LIN {X 0,Y 397.089,Z 381.624,A -85,B 0,C 180,E1 -11120.42,E2 -11120.42} C_VEL
LIN {X 0,Y 397.097,Z 381.645,A -85,B 0,C 180,E1 -11123.005,E2 -11123.005} C_VEL
LIN {X 0,Y 397.114,Z 381.63,A -85,B 0,C 180,E1 -11126.727,E2 -11126.727} C_VEL
LIN {X 0,Y 397.12,Z 381.643,A -85,B 0,C 180,E1 -11130.295,E2 -11130.295} C_VEL
LIN {X 0,Y 397.076,Z 381.648,A -85,B 0,C 180,E1 -11133.737,E2 -11133.737} C_VEL
LIN {X 0,Y 397.149,Z 381.85,A -85,B 0,C 180,E1 -11134.804,E2 -11134.804} C_VEL
LIN {X 0,Y 398.52,Z 387.762,A -85,B 0,C 180,E1 -11136.032,E2 -11136.032} C_VEL
LIN {X 0,Y 406.526,Z 408.883,A -85,B 0,C 180,E1 -11136.981,E2 -11136.981} C_VEL
LIN {X 0,Y 404.185,Z 503.873,A -85,B 0,C 180,E1 -11139.084,E2 -11139.084} C_VEL
LIN {X 0,Y 403.629,Z 530.739,A -85,B 0,C 180,E1 -11139.707,E2 -11139.707} C_VEL
LIN {X 0,Y 403.24,Z 546.56,A -85,B 0,C 180,E1 -11140.291,E2 -11140.291} C_VEL
LIN {X 0,Y 402.743,Z 560.989,A -85,B 0,C 180,E1 -11141.034,E2 -11141.034} C_VEL
LIN {X 0,Y 402.067,Z 574.399,A -85,B 0,C 180,E1 -11141.925,E2 -11141.925} C_VEL
LIN {X 0,Y 401.478,Z 586.705,A -85,B 0,C 180,E1 -11142.949,E2 -11142.949} C_VEL
LIN {X 0,Y 400.667,Z 599.243,A -85,B 0,C 180,E1 -11144.224,E2 -11144.224} C_VEL
LIN {X 0,Y 399.964,Z 610.425,A -85,B 0,C 180,E1 -11145.604,E2 -11145.604} C_VEL
LIN {X 0,Y 399.225,Z 620.083,A -85,B 0,C 180,E1 -11147.029,E2 -11147.029} C_VEL
LIN {X 0,Y 398.678,Z 628.735,A -85,B 0,C 180,E1 -11148.561,E2 -11148.561} C_VEL
LIN {X 0,Y 398.179,Z 637.057,A -85,B 0,C 180,E1 -11150.347,E2 -11150.347} C_VEL
LIN {X 0,Y 397.823,Z 642.855,A -85,B 0,C 180,E1 -11151.875,E2 -11151.875} C_VEL
LIN {X 0,Y 397.588,Z 647.629,A -85,B 0,C 180,E1 -11153.402,E2 -11153.402} C_VEL
LIN {X 0,Y 397.252,Z 651.509,A -85,B 0,C 180,E1 -11154.925,E2 -11154.925} C_VEL
LIN {X 0,Y 397.11,Z 653.565,A -85,B 0,C 180,E1 -11155.94,E2 -11155.94} C_VEL
LIN {X 0,Y 397.246,Z 655.212,A -85,B 0,C 180,E1 -11156.957,E2 -11156.957} C_VEL
LIN {X 0,Y 397.195,Z 657.492,A -85,B 0,C 180,E1 -11158.986,E2 -11158.986} C_VEL
LIN {X 0,Y 397.255,Z 658.37,A -85,B 0,C 180,E1 -11161.014,E2 -11161.014} C_VEL
LIN {X 0,Y 397.563,Z 657.822,A -85,B 0,C 180,E1 -11163.04,E2 -11163.04} C_VEL
LIN {X 0,Y 397.875,Z 655.889,A -85,B 0,C 180,E1 -11165.067,E2 -11165.067} C_VEL
LIN {X 0,Y 398.072,Z 654.383,A -85,B 0,C 180,E1 -11166.081,E2 -11166.081} C_VEL
LIN {X 0,Y 398.686,Z 651.307,A -85,B 0,C 180,E1 -11167.597,E2 -11167.597} C_VEL
LIN {X 0,Y 399.26,Z 646.78,A -85,B 0,C 180,E1 -11169.32,E2 -11169.32} C_VEL
LIN {X 0,Y 400.073,Z 640.589,A -85,B 0,C 180,E1 -11171.142,E2 -11171.142} C_VEL
LIN {X 0,Y 401.076,Z 633.002,A -85,B 0,C 180,E1 -11172.91,E2 -11172.91} C_VEL
LIN {X 0,Y 402.077,Z 624.982,A -85,B 0,C 180,E1 -11174.423,E2 -11174.423} C_VEL
LIN {X 0,Y 403.151,Z 615.267,A -85,B 0,C 180,E1 -11175.936,E2 -11175.936} C_VEL
LIN {X 0,Y 404.407,Z 603.369,A -85,B 0,C 180,E1 -11177.444,E2 -11177.444} C_VEL
LIN {X 0,Y 405.456,Z 591.237,A -85,B 0,C 180,E1 -11178.703,E2 -11178.703} C_VEL
LIN {X 0,Y 406.37,Z 579.301,A -85,B 0,C 180,E1 -11179.709,E2 -11179.709} C_VEL
LIN {X 0,Y 407.245,Z 566.122,A -85,B 0,C 180,E1 -11180.602,E2 -11180.602} C_VEL
LIN {X 0,Y 407.975,Z 552.389,A -85,B 0,C 180,E1 -11181.325,E2 -11181.325} C_VEL
LIN {X 0,Y 408.412,Z 537.34,A -85,B 0,C 180,E1 -11181.913,E2 -11181.913} C_VEL
LIN {X 0,Y 410.593,Z 491.111,A -85,B 0,C 180,E1 -11183.217,E2 -11183.217} C_VEL
LIN {X 0,Y 415.197,Z 422.298,A -85,B 0,C 180,E1 -11185.198,E2 -11185.198} C_VEL
LIN {X 0,Y 414.865,Z 420.892,A -85,B 0,C 180,E1 -11185.293,E2 -11185.293} C_VEL
LIN {X 0,Y 408.921,Z 410.512,A -85,B 0,C 180,E1 -11186.453,E2 -11186.453} C_VEL
LIN {X 0,Y 405.011,Z 404.284,A -85,B 0,C 180,E1 -11187.301,E2 -11187.301} C_VEL
LIN {X 0,Y 403.247,Z 398.209,A -85,B 0,C 180,E1 -11189.782,E2 -11189.782} C_VEL
LIN {X 0,Y 401.316,Z 392.497,A -85,B 0,C 180,E1 -11192.795,E2 -11192.795} C_VEL
LIN {X 0,Y 400.112,Z 388.952,A -85,B 0,C 180,E1 -11195.426,E2 -11195.426} C_VEL
LIN {X 0,Y 399.12,Z 386.996,A -85,B 0,C 180,E1 -11198.047,E2 -11198.047} C_VEL
LIN {X 0,Y 398.976,Z 386.521,A -85,B 0,C 180,E1 -11199.356,E2 -11199.356} C_VEL
LIN {X 0,Y 398.969,Z 386.501,A -85,B 0,C 180,E1 -11200.758,E2 -11200.758} C_VEL
LIN {X 0,Y 399.211,Z 387.025,A -85,B 0,C 180,E1 -11202.318,E2 -11202.318} C_VEL
LIN {X 0,Y 400.18,Z 388.851,A -85,B 0,C 180,E1 -11204.626,E2 -11204.626} C_VEL
LIN {X 0,Y 401.605,Z 392.32,A -85,B 0,C 180,E1 -11206.96,E2 -11206.96} C_VEL
LIN {X 0,Y 403.759,Z 397.673,A -85,B 0,C 180,E1 -11209.425,E2 -11209.425} C_VEL
LIN {X 0,Y 405.909,Z 403.521,A -85,B 0,C 180,E1 -11211.44,E2 -11211.44} C_VEL
LIN {X 0,Y 408.329,Z 411.193,A -85,B 0,C 180,E1 -11213.575,E2 -11213.575} C_VEL
LIN {X 0,Y 410.262,Z 418.651,A -85,B 0,C 180,E1 -11215.312,E2 -11215.312} C_VEL
LIN {X 0,Y 411.173,Z 423.227,A -85,B 0,C 180,E1 -11216.253,E2 -11216.253} C_VEL
LIN {X 0,Y 410.818,Z 426.707,A -85,B 0,C 180,E1 -11216.808,E2 -11216.808} C_VEL
LIN {X 0,Y 407.511,Z 447.425,A -85,B 0,C 180,E1 -11219.787,E2 -11219.787} C_VEL
LIN {X 0,Y 407.066,Z 451.037,A -85,B 0,C 180,E1 -11220.274,E2 -11220.274} C_VEL
LIN {X 0,Y 409.714,Z 468.904,A -85,B 0,C 180,E1 -11221.206,E2 -11221.206} C_VEL
LIN {X 0,Y 411.359,Z 484.62,A -85,B 0,C 180,E1 -11221.892,E2 -11221.892} C_VEL
LIN {X 0,Y 412.406,Z 501.199,A -85,B 0,C 180,E1 -11222.511,E2 -11222.511} C_VEL
LIN {X 0,Y 410.024,Z 555.027,A -85,B 0,C 180,E1 -11223.842,E2 -11223.842} C_VEL
LIN {X 0,Y 408.208,Z 641.314,A -85,B 0,C 180,E1 -11225.389,E2 -11225.389} C_VEL
LIN {X 0,Y 407.512,Z 656.884,A -85,B 0,C 180,E1 -11225.87,E2 -11225.87} C_VEL
LIN {X 0,Y 406.506,Z 672.375,A -85,B 0,C 180,E1 -11226.568,E2 -11226.568} C_VEL
LIN {X 0,Y 405.354,Z 686.866,A -85,B 0,C 180,E1 -11227.442,E2 -11227.442} C_VEL
LIN {X 0,Y 404.081,Z 700.048,A -85,B 0,C 180,E1 -11228.442,E2 -11228.442} C_VEL
LIN {X 0,Y 402.632,Z 713.43,A -85,B 0,C 180,E1 -11229.7,E2 -11229.7} C_VEL
LIN {X 0,Y 401.283,Z 725.191,A -85,B 0,C 180,E1 -11231.04,E2 -11231.04} C_VEL
LIN {X 0,Y 399.941,Z 736.663,A -85,B 0,C 180,E1 -11232.617,E2 -11232.617} C_VEL
LIN {X 0,Y 398.771,Z 747.384,A -85,B 0,C 180,E1 -11234.408,E2 -11234.408} C_VEL
LIN {X 0,Y 397.723,Z 756.499,A -85,B 0,C 180,E1 -11236.246,E2 -11236.246} C_VEL
LIN {X 0,Y 397.007,Z 764.608,A -85,B 0,C 180,E1 -11238.252,E2 -11238.252} C_VEL
LIN {X 0,Y 396.384,Z 771.265,A -85,B 0,C 180,E1 -11240.302,E2 -11240.302} C_VEL
LIN {X 0,Y 396.048,Z 776.466,A -85,B 0,C 180,E1 -11242.35,E2 -11242.35} C_VEL
LIN {X 0,Y 395.949,Z 779.458,A -85,B 0,C 180,E1 -11243.885,E2 -11243.885} C_VEL
LIN {X 0,Y 395.81,Z 782.389,A -85,B 0,C 180,E1 -11245.926,E2 -11245.926} C_VEL
LIN {X 0,Y 395.823,Z 784.133,A -85,B 0,C 180,E1 -11247.963,E2 -11247.963} C_VEL
LIN {X 0,Y 395.812,Z 784.728,A -85,B 0,C 180,E1 -11249.998,E2 -11249.998} C_VEL
LIN {X 0,Y 395.839,Z 784.13,A -85,B 0,C 180,E1 -11252.033,E2 -11252.033} C_VEL
LIN {X 0,Y 395.814,Z 782.381,A -85,B 0,C 180,E1 -11254.071,E2 -11254.071} C_VEL
LIN {X 0,Y 395.911,Z 779.235,A -85,B 0,C 180,E1 -11256.238,E2 -11256.238} C_VEL
LIN {X 0,Y 396.129,Z 775.273,A -85,B 0,C 180,E1 -11258.158,E2 -11258.158} C_VEL
LIN {X 0,Y 396.472,Z 769.727,A -85,B 0,C 180,E1 -11260.209,E2 -11260.209} C_VEL
LIN {X 0,Y 397.186,Z 762.664,A -85,B 0,C 180,E1 -11262.257,E2 -11262.257} C_VEL
LIN {X 0,Y 397.854,Z 755.214,A -85,B 0,C 180,E1 -11264.029,E2 -11264.029} C_VEL
LIN {X 0,Y 398.858,Z 745.957,A -85,B 0,C 180,E1 -11265.848,E2 -11265.848} C_VEL
LIN {X 0,Y 399.907,Z 736.641,A -85,B 0,C 180,E1 -11267.381,E2 -11267.381} C_VEL
LIN {X 0,Y 401.058,Z 727.016,A -85,B 0,C 180,E1 -11268.716,E2 -11268.716} C_VEL
LIN {X 0,Y 402.339,Z 715.741,A -85,B 0,C 180,E1 -11270.046,E2 -11270.046} C_VEL
LIN {X 0,Y 403.723,Z 702.844,A -85,B 0,C 180,E1 -11271.307,E2 -11271.307} C_VEL
LIN {X 0,Y 404.986,Z 690.311,A -85,B 0,C 180,E1 -11272.308,E2 -11272.308} C_VEL
LIN {X 0,Y 406.228,Z 675.667,A -85,B 0,C 180,E1 -11273.243,E2 -11273.243} C_VEL
LIN {X 0,Y 407.212,Z 661.406,A -85,B 0,C 180,E1 -11273.94,E2 -11273.94} C_VEL
LIN {X 0,Y 407.963,Z 646.864,A -85,B 0,C 180,E1 -11274.454,E2 -11274.454} C_VEL
LIN {X 0,Y 408.469,Z 630.141,A -85,B 0,C 180,E1 -11274.828,E2 -11274.828} C_VEL
LIN {X 0,Y 410.947,Z 500.531,A -85,B 0,C 180,E1 -11277.127,E2 -11277.127} C_VEL
LIN {X 0,Y 407.131,Z 470.69,A -85,B 0,C 180,E1 -11277.985,E2 -11277.985} C_VEL
LIN {X 0,Y 406.3,Z 464.366,A -85,B 0,C 180,E1 -11278.213,E2 -11278.213} C_VEL
LIN {X 0,Y 405.055,Z 449.15,A -85,B 0,C 180,E1 -11279.028,E2 -11279.028} C_VEL
LIN {X 0,Y 407.471,Z 422.518,A -85,B 0,C 180,E1 -11282.32,E2 -11282.32} C_VEL
LIN {X 0,Y 407.781,Z 419.227,A -85,B 0,C 180,E1 -11282.732,E2 -11282.732} C_VEL
LIN {X 0,Y 404.459,Z 406.774,A -85,B 0,C 180,E1 -11284.594,E2 -11284.594} C_VEL
LIN {X 0,Y 398.163,Z 385.398,A -85,B 0,C 180,E1 -11287.984,E2 -11287.984} C_VEL
LIN {X 0,Y 397.122,Z 381.788,A -85,B 0,C 180,E1 -11288.623,E2 -11288.623} C_VEL
LIN {X 0,Y 397.045,Z 381.654,A -85,B 0,C 180,E1 -11292.267,E2 -11292.267} C_VEL
LIN {X 0,Y 397.072,Z 381.648,A -85,B 0,C 180,E1 -11295.068,E2 -11295.068} C_VEL
LIN {X 0,Y 397.038,Z 381.618,A -85,B 0,C 180,E1 -11298.023,E2 -11298.023} C_VEL
LIN {X 0,Y 397.076,Z 381.648,A -85,B 0,C 180,E1 -11301.722,E2 -11301.722} C_VEL
LIN {X 0,Y 397.102,Z 381.606,A -85,B 0,C 180,E1 -11305.505,E2 -11305.505} C_VEL
LIN {X 0,Y 397.063,Z 381.648,A -85,B 0,C 180,E1 -11309.116,E2 -11309.116} C_VEL
LIN {X 0,Y 397.064,Z 381.647,A -85,B 0,C 180,E1 -11312.246,E2 -11312.246} C_VEL
LIN {X 0,Y 397.089,Z 381.633,A -85,B 0,C 180,E1 -11314.864,E2 -11314.864} C_VEL
LIN {X 0,Y 397.08,Z 381.65,A -85,B 0,C 180,E1 -11318.181,E2 -11318.181} C_VEL
LIN {X 0,Y 397.098,Z 381.641,A -85,B 0,C 180,E1 -11321.424,E2 -11321.424} C_VEL
LIN {X 0,Y 397.108,Z 381.631,A -85,B 0,C 180,E1 -11324.605,E2 -11324.605} C_VEL
LIN {X 0,Y 397.202,Z 381.631,A -85,B 0,C 180,E1 -11327.741,E2 -11327.741} C_VEL
LIN {X 0,Y 397.212,Z 381.618,A -85,B 0,C 180,E1 -11330.837,E2 -11330.837} C_VEL
LIN {X 0,Y 397.299,Z 381.618,A -85,B 0,C 180,E1 -11333.907,E2 -11333.907} C_VEL
LIN {X 0,Y 397.427,Z 381.601,A -85,B 0,C 180,E1 -11337.973,E2 -11337.973} C_VEL
LIN {X 0,Y 397.424,Z 381.591,A -85,B 0,C 180,E1 -11342.027,E2 -11342.027} C_VEL
LIN {X 0,Y 397.305,Z 381.606,A -85,B 0,C 180,E1 -11346.708,E2 -11346.708} C_VEL
LIN {X 0,Y 397.217,Z 381.629,A -85,B 0,C 180,E1 -11349.163,E2 -11349.163} C_VEL
LIN {X 0,Y 397.202,Z 381.616,A -85,B 0,C 180,E1 -11352.259,E2 -11352.259} C_VEL
LIN {X 0,Y 397.162,Z 381.629,A -85,B 0,C 180,E1 -11355.393,E2 -11355.393} C_VEL
LIN {X 0,Y 397.143,Z 381.638,A -85,B 0,C 180,E1 -11358.574,E2 -11358.574} C_VEL
LIN {X 0,Y 397.08,Z 381.638,A -85,B 0,C 180,E1 -11361.82,E2 -11361.82} C_VEL
LIN {X 0,Y 397.087,Z 381.636,A -85,B 0,C 180,E1 -11365.136,E2 -11365.136} C_VEL
LIN {X 0,Y 397.048,Z 381.648,A -85,B 0,C 180,E1 -11368.55,E2 -11368.55} C_VEL
LIN {X 0,Y 397.064,Z 381.649,A -85,B 0,C 180,E1 -11371.836,E2 -11371.836} C_VEL
LIN {X 0,Y 397.104,Z 381.649,A -85,B 0,C 180,E1 -11374.496,E2 -11374.496} C_VEL
LIN {X 0,Y 397.077,Z 381.623,A -85,B 0,C 180,E1 -11378.278,E2 -11378.278} C_VEL
LIN {X 0,Y 397.035,Z 381.648,A -85,B 0,C 180,E1 -11380.916,E2 -11380.916} C_VEL
LIN {X 0,Y 397.075,Z 381.635,A -85,B 0,C 180,E1 -11383.652,E2 -11383.652} C_VEL
LIN {X 0,Y 397.08,Z 381.631,A -85,B 0,C 180,E1 -11386.525,E2 -11386.525} C_VEL
LIN {X 0,Y 397.13,Z 381.847,A -85,B 0,C 180,E1 -11389.321,E2 -11389.321} C_VEL
LIN {X 0,Y 399.981,Z 390.021,A -85,B 0,C 180,E1 -11390.764,E2 -11390.764} C_VEL
LIN {X 0,Y 405.051,Z 405.352,A -85,B 0,C 180,E1 -11393.294,E2 -11393.294} C_VEL
LIN {X 0,Y 409.446,Z 421.082,A -85,B 0,C 180,E1 -11395.744,E2 -11395.744} C_VEL
LIN {X 0,Y 409.79,Z 422.39,A -85,B 0,C 180,E1 -11395.94,E2 -11395.94} C_VEL
LIN {X 0,Y 409.04,Z 433.785,A -85,B 0,C 180,E1 -11397.342,E2 -11397.342} C_VEL
LIN {X 0,Y 407.476,Z 457.22,A -85,B 0,C 180,E1 -11400.133,E2 -11400.133} C_VEL
LIN {X 0,Y 406.73,Z 471.528,A -85,B 0,C 180,E1 -11401.751,E2 -11401.751} C_VEL
LIN {X 0,Y 411.653,Z 502.312,A -85,B 0,C 180,E1 -11402.733,E2 -11402.733} C_VEL
LIN {X 0,Y 408.849,Z 639.721,A -85,B 0,C 180,E1 -11405.197,E2 -11405.197} C_VEL
LIN {X 0,Y 408.137,Z 655.686,A -85,B 0,C 180,E1 -11405.665,E2 -11405.665} C_VEL
LIN {X 0,Y 407.159,Z 670.76,A -85,B 0,C 180,E1 -11406.317,E2 -11406.317} C_VEL
LIN {X 0,Y 406.104,Z 684.154,A -85,B 0,C 180,E1 -11407.086,E2 -11407.086} C_VEL
LIN {X 0,Y 404.743,Z 697.956,A -85,B 0,C 180,E1 -11408.081,E2 -11408.081} C_VEL
LIN {X 0,Y 403.391,Z 710.624,A -85,B 0,C 180,E1 -11409.21,E2 -11409.21} C_VEL
LIN {X 0,Y 402.084,Z 722.357,A -85,B 0,C 180,E1 -11410.473,E2 -11410.473} C_VEL
LIN {X 0,Y 400.806,Z 733.238,A -85,B 0,C 180,E1 -11411.868,E2 -11411.868} C_VEL
LIN {X 0,Y 399.525,Z 743.27,A -85,B 0,C 180,E1 -11413.392,E2 -11413.392} C_VEL
LIN {X 0,Y 398.336,Z 753.073,A -85,B 0,C 180,E1 -11415.179,E2 -11415.179} C_VEL
LIN {X 0,Y 397.433,Z 761.858,A -85,B 0,C 180,E1 -11417.133,E2 -11417.133} C_VEL
LIN {X 0,Y 396.459,Z 764.8,A -85,B 0,C 180,E1 -11417.861,E2 -11417.861} C_VEL
LIN {X 0,Y 393.176,Z 769.275,A -85,B 0,C 180,E1 -11419.057,E2 -11419.057} C_VEL
LIN {X 0,Y 389.974,Z 773.232,A -85,B 0,C 180,E1 -11420.305,E2 -11420.305} C_VEL
LIN {X 0,Y 389.137,Z 775.372,A -85,B 0,C 180,E1 -11421.103,E2 -11421.103} C_VEL
LIN {X 0,Y 388.85,Z 779.022,A -85,B 0,C 180,E1 -11422.733,E2 -11422.733} C_VEL
LIN {X 0,Y 388.697,Z 782.564,A -85,B 0,C 180,E1 -11424.815,E2 -11424.815} C_VEL
LIN {X 0,Y 388.59,Z 784.906,A -85,B 0,C 180,E1 -11426.891,E2 -11426.891} C_VEL
LIN {X 0,Y 388.652,Z 786.099,A -85,B 0,C 180,E1 -11428.965,E2 -11428.965} C_VEL
LIN {X 0,Y 388.653,Z 786.114,A -85,B 0,C 180,E1 -11431.038,E2 -11431.038} C_VEL
LIN {X 0,Y 388.591,Z 784.981,A -85,B 0,C 180,E1 -11433.112,E2 -11433.112} C_VEL
LIN {X 0,Y 388.709,Z 782.697,A -85,B 0,C 180,E1 -11435.188,E2 -11435.188} C_VEL
LIN {X 0,Y 388.919,Z 779.209,A -85,B 0,C 180,E1 -11437.269,E2 -11437.269} C_VEL
LIN {X 0,Y 389.212,Z 774.436,A -85,B 0,C 180,E1 -11439.354,E2 -11439.354} C_VEL
LIN {X 0,Y 389.809,Z 768.258,A -85,B 0,C 180,E1 -11441.44,E2 -11441.44} C_VEL
LIN {X 0,Y 390.607,Z 760.487,A -85,B 0,C 180,E1 -11443.528,E2 -11443.528} C_VEL
LIN {X 0,Y 391.54,Z 752.198,A -85,B 0,C 180,E1 -11445.354,E2 -11445.354} C_VEL
LIN {X 0,Y 392.795,Z 742.215,A -85,B 0,C 180,E1 -11447.172,E2 -11447.172} C_VEL
LIN {X 0,Y 394.141,Z 732.023,A -85,B 0,C 180,E1 -11448.722,E2 -11448.722} C_VEL
LIN {X 0,Y 395.612,Z 719.815,A -85,B 0,C 180,E1 -11450.27,E2 -11450.27} C_VEL
LIN {X 0,Y 397.133,Z 707.618,A -85,B 0,C 180,E1 -11451.545,E2 -11451.545} C_VEL
LIN {X 0,Y 398.532,Z 694.315,A -85,B 0,C 180,E1 -11452.692,E2 -11452.692} C_VEL
LIN {X 0,Y 399.989,Z 679.521,A -85,B 0,C 180,E1 -11453.7,E2 -11453.7} C_VEL
LIN {X 0,Y 401.097,Z 664.893,A -85,B 0,C 180,E1 -11454.472,E2 -11454.472} C_VEL
LIN {X 0,Y 402.017,Z 649.798,A -85,B 0,C 180,E1 -11455.05,E2 -11455.05} C_VEL
LIN {X 0,Y 402.559,Z 634.992,A -85,B 0,C 180,E1 -11455.429,E2 -11455.429} C_VEL
LIN {X 0,Y 405.369,Z 503.814,A -85,B 0,C 180,E1 -11457.794,E2 -11457.794} C_VEL
LIN {X 0,Y 400.361,Z 472.201,A -85,B 0,C 180,E1 -11458.805,E2 -11458.805} C_VEL
LIN {X 0,Y 400.3,Z 469.804,A -85,B 0,C 180,E1 -11459.02,E2 -11459.02} C_VEL
LIN {X 0,Y 401.927,Z 444.921,A -85,B 0,C 180,E1 -11461.935,E2 -11461.935} C_VEL
LIN {X 0,Y 403.408,Z 425.683,A -85,B 0,C 180,E1 -11464.296,E2 -11464.296} C_VEL
LIN {X 0,Y 400.308,Z 413.802,A -85,B 0,C 180,E1 -11466.138,E2 -11466.138} C_VEL
LIN {X 0,Y 395.695,Z 398.735,A -85,B 0,C 180,E1 -11468.602,E2 -11468.602} C_VEL
LIN {X 0,Y 390.413,Z 384.107,A -85,B 0,C 180,E1 -11471.156,E2 -11471.156} C_VEL
LIN {X 0,Y 390.024,Z 382.673,A -85,B 0,C 180,E1 -11471.479,E2 -11471.479} C_VEL
LIN {X 0,Y 390.008,Z 382.518,A -85,B 0,C 180,E1 -11474.652,E2 -11474.652} C_VEL
LIN {X 0,Y 390.03,Z 382.528,A -85,B 0,C 180,E1 -11477.629,E2 -11477.629} C_VEL
LIN {X 0,Y 390.059,Z 382.504,A -85,B 0,C 180,E1 -11480.904,E2 -11480.904} C_VEL
LIN {X 0,Y 390.072,Z 382.494,A -85,B 0,C 180,E1 -11484.792,E2 -11484.792} C_VEL
LIN {X 0,Y 390.022,Z 382.527,A -85,B 0,C 180,E1 -11488.495,E2 -11488.495} C_VEL
LIN {X 0,Y 390.021,Z 382.528,A -85,B 0,C 180,E1 -11492.003,E2 -11492.003} C_VEL
LIN {X 0,Y 390.076,Z 382.707,A -85,B 0,C 180,E1 -11494.469,E2 -11494.469} C_VEL
LIN {X 0,Y 391.413,Z 388.26,A -85,B 0,C 180,E1 -11495.65,E2 -11495.65} C_VEL
LIN {X 0,Y 399.879,Z 410.632,A -85,B 0,C 180,E1 -11496.682,E2 -11496.682} C_VEL
LIN {X 0,Y 397.151,Z 511.569,A -85,B 0,C 180,E1 -11498.967,E2 -11498.967} C_VEL
LIN {X 0,Y 396.771,Z 533.461,A -85,B 0,C 180,E1 -11499.518,E2 -11499.518} C_VEL
LIN {X 0,Y 396.367,Z 548.749,A -85,B 0,C 180,E1 -11500.114,E2 -11500.114} C_VEL
LIN {X 0,Y 395.802,Z 563.167,A -85,B 0,C 180,E1 -11500.89,E2 -11500.89} C_VEL
LIN {X 0,Y 395.081,Z 577.072,A -85,B 0,C 180,E1 -11501.862,E2 -11501.862} C_VEL
LIN {X 0,Y 394.386,Z 590.414,A -85,B 0,C 180,E1 -11503.034,E2 -11503.034} C_VEL
LIN {X 0,Y 393.54,Z 602.523,A -85,B 0,C 180,E1 -11504.329,E2 -11504.329} C_VEL
LIN {X 0,Y 392.896,Z 613.545,A -85,B 0,C 180,E1 -11505.762,E2 -11505.762} C_VEL
LIN {X 0,Y 392.088,Z 623.491,A -85,B 0,C 180,E1 -11507.316,E2 -11507.316} C_VEL
LIN {X 0,Y 391.581,Z 631.771,A -85,B 0,C 180,E1 -11508.876,E2 -11508.876} C_VEL
LIN {X 0,Y 391.054,Z 639.69,A -85,B 0,C 180,E1 -11510.692,E2 -11510.692} C_VEL
LIN {X 0,Y 390.797,Z 645.268,A -85,B 0,C 180,E1 -11512.248,E2 -11512.248} C_VEL
LIN {X 0,Y 390.406,Z 651.086,A -85,B 0,C 180,E1 -11514.318,E2 -11514.318} C_VEL
LIN {X 0,Y 390.084,Z 654.454,A -85,B 0,C 180,E1 -11515.867,E2 -11515.867} C_VEL
LIN {X 0,Y 390.224,Z 656.151,A -85,B 0,C 180,E1 -11516.903,E2 -11516.903} C_VEL
LIN {X 0,Y 390.172,Z 658.517,A -85,B 0,C 180,E1 -11518.968,E2 -11518.968} C_VEL
LIN {X 0,Y 390.265,Z 659.479,A -85,B 0,C 180,E1 -11521.032,E2 -11521.032} C_VEL
LIN {X 0,Y 390.595,Z 659.016,A -85,B 0,C 180,E1 -11523.094,E2 -11523.094} C_VEL
LIN {X 0,Y 390.933,Z 657.159,A -85,B 0,C 180,E1 -11525.157,E2 -11525.157} C_VEL
LIN {X 0,Y 391.53,Z 653.812,A -85,B 0,C 180,E1 -11527.218,E2 -11527.218} C_VEL
LIN {X 0,Y 392.184,Z 650.228,A -85,B 0,C 180,E1 -11528.761,E2 -11528.761} C_VEL
LIN {X 0,Y 393.006,Z 644.059,A -85,B 0,C 180,E1 -11530.822,E2 -11530.822} C_VEL
LIN {X 0,Y 394.052,Z 636.985,A -85,B 0,C 180,E1 -11532.62,E2 -11532.62} C_VEL
LIN {X 0,Y 395.032,Z 629.546,A -85,B 0,C 180,E1 -11534.16,E2 -11534.16} C_VEL
LIN {X 0,Y 396.141,Z 620.614,A -85,B 0,C 180,E1 -11535.697,E2 -11535.697} C_VEL
LIN {X 0,Y 397.418,Z 610.224,A -85,B 0,C 180,E1 -11537.159,E2 -11537.159} C_VEL
LIN {X 0,Y 398.573,Z 598.641,A -85,B 0,C 180,E1 -11538.505,E2 -11538.505} C_VEL
LIN {X 0,Y 399.734,Z 585.186,A -85,B 0,C 180,E1 -11539.782,E2 -11539.782} C_VEL
LIN {X 0,Y 400.789,Z 571.82,A -85,B 0,C 180,E1 -11540.779,E2 -11540.779} C_VEL
LIN {X 0,Y 401.565,Z 558.555,A -85,B 0,C 180,E1 -11541.563,E2 -11541.563} C_VEL
LIN {X 0,Y 402.225,Z 543.117,A -85,B 0,C 180,E1 -11542.247,E2 -11542.247} C_VEL
LIN {X 0,Y 402.947,Z 523.32,A -85,B 0,C 180,E1 -11542.868,E2 -11542.868} C_VEL
LIN {X 0,Y 407.69,Z 450.848,A -85,B 0,C 180,E1 -11544.986,E2 -11544.986} C_VEL
LIN {X 0,Y 409.599,Z 424.289,A -85,B 0,C 180,E1 -11545.798,E2 -11545.798} C_VEL
LIN {X 0,Y 403.85,Z 414.342,A -85,B 0,C 180,E1 -11546.98,E2 -11546.98} C_VEL
LIN {X 0,Y 399.918,Z 408.279,A -85,B 0,C 180,E1 -11547.856,E2 -11547.856} C_VEL
LIN {X 0,Y 398.459,Z 405.901,A -85,B 0,C 180,E1 -11548.245,E2 -11548.245} C_VEL
LIN {X 0,Y 397.356,Z 402.068,A -85,B 0,C 180,E1 -11549.926,E2 -11549.926} C_VEL
LIN {X 0,Y 395.951,Z 397.866,A -85,B 0,C 180,E1 -11552.174,E2 -11552.174} C_VEL
LIN {X 0,Y 394.762,Z 394.232,A -85,B 0,C 180,E1 -11554.729,E2 -11554.729} C_VEL
LIN {X 0,Y 394.075,Z 392.435,A -85,B 0,C 180,E1 -11556.625,E2 -11556.625} C_VEL
LIN {X 0,Y 393.634,Z 391.377,A -85,B 0,C 180,E1 -11558.674,E2 -11558.674} C_VEL
LIN {X 0,Y 393.579,Z 391.134,A -85,B 0,C 180,E1 -11560.004,E2 -11560.004} C_VEL
LIN {X 0,Y 393.672,Z 391.35,A -85,B 0,C 180,E1 -11561.425,E2 -11561.425} C_VEL
LIN {X 0,Y 394.105,Z 392.188,A -85,B 0,C 180,E1 -11563.016,E2 -11563.016} C_VEL
LIN {X 0,Y 394.874,Z 393.548,A -85,B 0,C 180,E1 -11564.607,E2 -11564.607} C_VEL
LIN {X 0,Y 396.056,Z 396.575,A -85,B 0,C 180,E1 -11566.681,E2 -11566.681} C_VEL
LIN {X 0,Y 397.663,Z 400.484,A -85,B 0,C 180,E1 -11568.662,E2 -11568.662} C_VEL
LIN {X 0,Y 399.588,Z 405.859,A -85,B 0,C 180,E1 -11570.714,E2 -11570.714} C_VEL
LIN {X 0,Y 401.754,Z 412.507,A -85,B 0,C 180,E1 -11572.744,E2 -11572.744} C_VEL
LIN {X 0,Y 403.97,Z 420.903,A -85,B 0,C 180,E1 -11574.852,E2 -11574.852} C_VEL
LIN {X 0,Y 405.017,Z 426.286,A -85,B 0,C 180,E1 -11576,E2 -11576} C_VEL
LIN {X 0,Y 403.544,Z 434.854,A -85,B 0,C 180,E1 -11577.323,E2 -11577.323} C_VEL
LIN {X 0,Y 401.139,Z 449.55,A -85,B 0,C 180,E1 -11579.462,E2 -11579.462} C_VEL
LIN {X 0,Y 403.996,Z 469.342,A -85,B 0,C 180,E1 -11580.572,E2 -11580.572} C_VEL
LIN {X 0,Y 405.613,Z 485.303,A -85,B 0,C 180,E1 -11581.303,E2 -11581.303} C_VEL
LIN {X 0,Y 406.6,Z 501.492,A -85,B 0,C 180,E1 -11581.941,E2 -11581.941} C_VEL
LIN {X 0,Y 403.448,Z 564.153,A -85,B 0,C 180,E1 -11583.556,E2 -11583.556} C_VEL
LIN {X 0,Y 401.772,Z 641.431,A -85,B 0,C 180,E1 -11584.968,E2 -11584.968} C_VEL
LIN {X 0,Y 401.027,Z 657.145,A -85,B 0,C 180,E1 -11585.462,E2 -11585.462} C_VEL
LIN {X 0,Y 400,Z 672.425,A -85,B 0,C 180,E1 -11586.163,E2 -11586.163} C_VEL
LIN {X 0,Y 398.807,Z 686.906,A -85,B 0,C 180,E1 -11587.05,E2 -11587.05} C_VEL
LIN {X 0,Y 397.476,Z 700.081,A -85,B 0,C 180,E1 -11588.066,E2 -11588.066} C_VEL
LIN {X 0,Y 395.956,Z 713.459,A -85,B 0,C 180,E1 -11589.342,E2 -11589.342} C_VEL
LIN {X 0,Y 394.458,Z 725.84,A -85,B 0,C 180,E1 -11590.785,E2 -11590.785} C_VEL
LIN {X 0,Y 393.131,Z 736.686,A -85,B 0,C 180,E1 -11592.306,E2 -11592.306} C_VEL
LIN {X 0,Y 391.859,Z 747.405,A -85,B 0,C 180,E1 -11594.125,E2 -11594.125} C_VEL
LIN {X 0,Y 390.797,Z 756.313,A -85,B 0,C 180,E1 -11595.948,E2 -11595.948} C_VEL
LIN {X 0,Y 390.189,Z 762.699,A -85,B 0,C 180,E1 -11597.516,E2 -11597.516} C_VEL
LIN {X 0,Y 389.433,Z 769.752,A -85,B 0,C 180,E1 -11599.602,E2 -11599.602} C_VEL
LIN {X 0,Y 389.068,Z 775.29,A -85,B 0,C 180,E1 -11601.69,E2 -11601.69} C_VEL
LIN {X 0,Y 388.873,Z 779.473,A -85,B 0,C 180,E1 -11603.773,E2 -11603.773} C_VEL
LIN {X 0,Y 388.734,Z 782.403,A -85,B 0,C 180,E1 -11605.851,E2 -11605.851} C_VEL
LIN {X 0,Y 388.72,Z 784.147,A -85,B 0,C 180,E1 -11607.926,E2 -11607.926} C_VEL
LIN {X 0,Y 388.74,Z 784.741,A -85,B 0,C 180,E1 -11609.998,E2 -11609.998} C_VEL
LIN {X 0,Y 388.735,Z 784.144,A -85,B 0,C 180,E1 -11612.071,E2 -11612.071} C_VEL
LIN {X 0,Y 388.736,Z 782.395,A -85,B 0,C 180,E1 -11614.145,E2 -11614.145} C_VEL
LIN {X 0,Y 388.831,Z 779.467,A -85,B 0,C 180,E1 -11616.224,E2 -11616.224} C_VEL
LIN {X 0,Y 389.062,Z 775.287,A -85,B 0,C 180,E1 -11618.307,E2 -11618.307} C_VEL
LIN {X 0,Y 389.426,Z 769.742,A -85,B 0,C 180,E1 -11620.395,E2 -11620.395} C_VEL
LIN {X 0,Y 390.185,Z 762.679,A -85,B 0,C 180,E1 -11622.481,E2 -11622.481} C_VEL
LIN {X 0,Y 390.899,Z 755.23,A -85,B 0,C 180,E1 -11624.284,E2 -11624.284} C_VEL
LIN {X 0,Y 391.978,Z 745.974,A -85,B 0,C 180,E1 -11626.134,E2 -11626.134} C_VEL
LIN {X 0,Y 393.111,Z 736.66,A -85,B 0,C 180,E1 -11627.692,E2 -11627.692} C_VEL
LIN {X 0,Y 394.427,Z 725.893,A -85,B 0,C 180,E1 -11629.202,E2 -11629.202} C_VEL
LIN {X 0,Y 395.928,Z 713.429,A -85,B 0,C 180,E1 -11630.656,E2 -11630.656} C_VEL
LIN {X 0,Y 397.454,Z 700.028,A -85,B 0,C 180,E1 -11631.932,E2 -11631.932} C_VEL
LIN {X 0,Y 398.749,Z 686.835,A -85,B 0,C 180,E1 -11632.95,E2 -11632.95} C_VEL
LIN {X 0,Y 399.963,Z 672.351,A -85,B 0,C 180,E1 -11633.836,E2 -11633.836} C_VEL
LIN {X 0,Y 401.016,Z 657.178,A -85,B 0,C 180,E1 -11634.529,E2 -11634.529} C_VEL
LIN {X 0,Y 401.733,Z 641.222,A -85,B 0,C 180,E1 -11635.031,E2 -11635.031} C_VEL
LIN {X 0,Y 404.172,Z 527.188,A -85,B 0,C 180,E1 -11637.102,E2 -11637.102} C_VEL
LIN {X 0,Y 404.491,Z 499.972,A -85,B 0,C 180,E1 -11637.61,E2 -11637.61} C_VEL
LIN {X 0,Y 400.607,Z 469.891,A -85,B 0,C 180,E1 -11638.501,E2 -11638.501} C_VEL
LIN {X 0,Y 399.869,Z 463.935,A -85,B 0,C 180,E1 -11638.731,E2 -11638.731} C_VEL
LIN {X 0,Y 398.546,Z 446.617,A -85,B 0,C 180,E1 -11639.692,E2 -11639.692} C_VEL
LIN {X 0,Y 400.989,Z 421.074,A -85,B 0,C 180,E1 -11642.908,E2 -11642.908} C_VEL
LIN {X 0,Y 398.213,Z 410.464,A -85,B 0,C 180,E1 -11644.519,E2 -11644.519} C_VEL
LIN {X 0,Y 392.002,Z 389.22,A -85,B 0,C 180,E1 -11647.922,E2 -11647.922} C_VEL
LIN {X 0,Y 390.055,Z 382.665,A -85,B 0,C 180,E1 -11649.069,E2 -11649.069} C_VEL
LIN {X 0,Y 390.021,Z 382.529,A -85,B 0,C 180,E1 -11652.371,E2 -11652.371} C_VEL
LIN {X 0,Y 390.028,Z 382.525,A -85,B 0,C 180,E1 -11655.352,E2 -11655.352} C_VEL
LIN {X 0,Y 390.001,Z 382.494,A -85,B 0,C 180,E1 -11658.183,E2 -11658.183} C_VEL
LIN {X 0,Y 390.044,Z 382.525,A -85,B 0,C 180,E1 -11660.902,E2 -11660.902} C_VEL
LIN {X 0,Y 390.054,Z 382.479,A -85,B 0,C 180,E1 -11664.79,E2 -11664.79} C_VEL
LIN {X 0,Y 390.009,Z 382.532,A -85,B 0,C 180,E1 -11668.494,E2 -11668.494} C_VEL
LIN {X 0,Y 390.011,Z 382.523,A -85,B 0,C 180,E1 -11672.062,E2 -11672.062} C_VEL
LIN {X 0,Y 390.028,Z 382.512,A -85,B 0,C 180,E1 -11675.516,E2 -11675.516} C_VEL
LIN {X 0,Y 390.04,Z 382.517,A -85,B 0,C 180,E1 -11678.877,E2 -11678.877} C_VEL
LIN {X 0,Y 390.052,Z 382.522,A -85,B 0,C 180,E1 -11682.163,E2 -11682.163} C_VEL
LIN {X 0,Y 390.076,Z 382.505,A -85,B 0,C 180,E1 -11685.39,E2 -11685.39} C_VEL
LIN {X 0,Y 390.154,Z 382.509,A -85,B 0,C 180,E1 -11687.516,E2 -11687.516} C_VEL
LIN {X 0,Y 390.171,Z 382.494,A -85,B 0,C 180,E1 -11690.671,E2 -11690.671} C_VEL
LIN {X 0,Y 390.255,Z 382.495,A -85,B 0,C 180,E1 -11693.797,E2 -11693.797} C_VEL
LIN {X 0,Y 390.394,Z 382.477,A -85,B 0,C 180,E1 -11697.937,E2 -11697.937} C_VEL
LIN {X 0,Y 390.391,Z 382.467,A -85,B 0,C 180,E1 -11702.063,E2 -11702.063} C_VEL
LIN {X 0,Y 390.259,Z 382.483,A -85,B 0,C 180,E1 -11706.704,E2 -11706.704} C_VEL
LIN {X 0,Y 390.174,Z 382.505,A -85,B 0,C 180,E1 -11709.33,E2 -11709.33} C_VEL
LIN {X 0,Y 390.154,Z 382.496,A -85,B 0,C 180,E1 -11712.484,E2 -11712.484} C_VEL
LIN {X 0,Y 390.123,Z 382.505,A -85,B 0,C 180,E1 -11715.678,E2 -11715.678} C_VEL
LIN {X 0,Y 390.088,Z 382.519,A -85,B 0,C 180,E1 -11718.923,E2 -11718.923} C_VEL
LIN {X 0,Y 390.02,Z 382.52,A -85,B 0,C 180,E1 -11722.235,E2 -11722.235} C_VEL
LIN {X 0,Y 390.036,Z 382.514,A -85,B 0,C 180,E1 -11725.723,E2 -11725.723} C_VEL
LIN {X 0,Y 390.009,Z 382.521,A -85,B 0,C 180,E1 -11729.114,E2 -11729.114} C_VEL
LIN {X 0,Y 390.027,Z 382.522,A -85,B 0,C 180,E1 -11732.723,E2 -11732.723} C_VEL
LIN {X 0,Y 390.03,Z 382.515,A -85,B 0,C 180,E1 -11735.824,E2 -11735.824} C_VEL
LIN {X 0,Y 390.024,Z 382.517,A -85,B 0,C 180,E1 -11739.213,E2 -11739.213} C_VEL
LIN {X 0,Y 390.018,Z 382.504,A -85,B 0,C 180,E1 -11742.373,E2 -11742.373} C_VEL
LIN {X 0,Y 390.029,Z 382.523,A -85,B 0,C 180,E1 -11745.355,E2 -11745.355} C_VEL
LIN {X 0,Y 390.033,Z 382.73,A -85,B 0,C 180,E1 -11748.669,E2 -11748.669} C_VEL
LIN {X 0,Y 392.64,Z 390.021,A -85,B 0,C 180,E1 -11750.012,E2 -11750.012} C_VEL
LIN {X 0,Y 397.877,Z 405.616,A -85,B 0,C 180,E1 -11752.643,E2 -11752.643} C_VEL
LIN {X 0,Y 401.707,Z 418.642,A -85,B 0,C 180,E1 -11754.738,E2 -11754.738} C_VEL
LIN {X 0,Y 403.329,Z 424.987,A -85,B 0,C 180,E1 -11755.716,E2 -11755.716} C_VEL
LIN {X 0,Y 401.836,Z 446.548,A -85,B 0,C 180,E1 -11758.355,E2 -11758.355} C_VEL
LIN {X 0,Y 400.257,Z 471.358,A -85,B 0,C 180,E1 -11761.246,E2 -11761.246} C_VEL
LIN {X 0,Y 405.313,Z 503.101,A -85,B 0,C 180,E1 -11762.287,E2 -11762.287} C_VEL
LIN {X 0,Y 402.417,Z 639.637,A -85,B 0,C 180,E1 -11764.773,E2 -11764.773} C_VEL
LIN {X 0,Y 401.662,Z 655.783,A -85,B 0,C 180,E1 -11765.253,E2 -11765.253} C_VEL
LIN {X 0,Y 400.643,Z 670.721,A -85,B 0,C 180,E1 -11765.907,E2 -11765.907} C_VEL
LIN {X 0,Y 399.545,Z 684.124,A -85,B 0,C 180,E1 -11766.688,E2 -11766.688} C_VEL
LIN {X 0,Y 398.141,Z 697.93,A -85,B 0,C 180,E1 -11767.698,E2 -11767.698} C_VEL
LIN {X 0,Y 396.74,Z 710.602,A -85,B 0,C 180,E1 -11768.845,E2 -11768.845} C_VEL
LIN {X 0,Y 395.362,Z 722.337,A -85,B 0,C 180,E1 -11770.127,E2 -11770.127} C_VEL
LIN {X 0,Y 394.017,Z 733.22,A -85,B 0,C 180,E1 -11771.544,E2 -11771.544} C_VEL
LIN {X 0,Y 392.683,Z 743.253,A -85,B 0,C 180,E1 -11773.094,E2 -11773.094} C_VEL
LIN {X 0,Y 391.436,Z 753.057,A -85,B 0,C 180,E1 -11774.912,E2 -11774.912} C_VEL
LIN {X 0,Y 390.535,Z 761.194,A -85,B 0,C 180,E1 -11776.737,E2 -11776.737} C_VEL
LIN {X 0,Y 389.824,Z 767.938,A -85,B 0,C 180,E1 -11778.563,E2 -11778.563} C_VEL
LIN {X 0,Y 389.24,Z 774.19,A -85,B 0,C 180,E1 -11780.65,E2 -11780.65} C_VEL
LIN {X 0,Y 389.137,Z 775.372,A -85,B 0,C 180,E1 -11781.103,E2 -11781.103} C_VEL
LIN {X 0,Y 388.319,Z 777.373,A -85,B 0,C 180,E1 -11781.914,E2 -11781.914} C_VEL
LIN {X 0,Y 385.249,Z 780.156,A -85,B 0,C 180,E1 -11783.25,E2 -11783.25} C_VEL
LIN {X 0,Y 382.727,Z 782.027,A -85,B 0,C 180,E1 -11784.347,E2 -11784.347} C_VEL
LIN {X 0,Y 381.662,Z 783.21,A -85,B 0,C 180,E1 -11785.205,E2 -11785.205} C_VEL
LIN {X 0,Y 381.582,Z 783.519,A -85,B 0,C 180,E1 -11785.497,E2 -11785.497} C_VEL
LIN {X 0,Y 381.51,Z 785.63,A -85,B 0,C 180,E1 -11787.89,E2 -11787.89} C_VEL
LIN {X 0,Y 381.54,Z 786.243,A -85,B 0,C 180,E1 -11790.002,E2 -11790.002} C_VEL
LIN {X 0,Y 381.511,Z 785.675,A -85,B 0,C 180,E1 -11792.113,E2 -11792.113} C_VEL
LIN {X 0,Y 381.593,Z 783.971,A -85,B 0,C 180,E1 -11794.226,E2 -11794.226} C_VEL
LIN {X 0,Y 381.71,Z 781.092,A -85,B 0,C 180,E1 -11796.344,E2 -11796.344} C_VEL
LIN {X 0,Y 381.969,Z 776.973,A -85,B 0,C 180,E1 -11798.466,E2 -11798.466} C_VEL
LIN {X 0,Y 382.386,Z 771.516,A -85,B 0,C 180,E1 -11800.592,E2 -11800.592} C_VEL
LIN {X 0,Y 383.181,Z 764.568,A -85,B 0,C 180,E1 -11802.716,E2 -11802.716} C_VEL
LIN {X 0,Y 384.024,Z 757.123,A -85,B 0,C 180,E1 -11804.576,E2 -11804.576} C_VEL
LIN {X 0,Y 385.201,Z 748.15,A -85,B 0,C 180,E1 -11806.429,E2 -11806.429} C_VEL
LIN {X 0,Y 386.425,Z 738.988,A -85,B 0,C 180,E1 -11808.011,E2 -11808.011} C_VEL
LIN {X 0,Y 387.967,Z 727.511,A -85,B 0,C 180,E1 -11809.675,E2 -11809.675} C_VEL
LIN {X 0,Y 389.533,Z 715.186,A -85,B 0,C 180,E1 -11811.153,E2 -11811.153} C_VEL
LIN {X 0,Y 391.113,Z 702.016,A -85,B 0,C 180,E1 -11812.449,E2 -11812.449} C_VEL
LIN {X 0,Y 392.569,Z 689.129,A -85,B 0,C 180,E1 -11813.475,E2 -11813.475} C_VEL
LIN {X 0,Y 393.852,Z 674.914,A -85,B 0,C 180,E1 -11814.386,E2 -11814.386} C_VEL
LIN {X 0,Y 394.915,Z 660.215,A -85,B 0,C 180,E1 -11815.105,E2 -11815.105} C_VEL
LIN {X 0,Y 395.882,Z 644.421,A -85,B 0,C 180,E1 -11815.642,E2 -11815.642} C_VEL
LIN {X 0,Y 396.386,Z 624.259,A -85,B 0,C 180,E1 -11816.065,E2 -11816.065} C_VEL
LIN {X 0,Y 399.08,Z 504.806,A -85,B 0,C 180,E1 -11818.248,E2 -11818.248} C_VEL
LIN {X 0,Y 394.195,Z 473.61,A -85,B 0,C 180,E1 -11819.265,E2 -11819.265} C_VEL
LIN {X 0,Y 393.814,Z 471.122,A -85,B 0,C 180,E1 -11819.388,E2 -11819.388} C_VEL
LIN {X 0,Y 395.339,Z 448.211,A -85,B 0,C 180,E1 -11822.081,E2 -11822.081} C_VEL
LIN {X 0,Y 396.876,Z 428.399,A -85,B 0,C 180,E1 -11824.519,E2 -11824.519} C_VEL
LIN {X 0,Y 396.205,Z 424.612,A -85,B 0,C 180,E1 -11825.085,E2 -11825.085} C_VEL
LIN {X 0,Y 391.36,Z 407.888,A -85,B 0,C 180,E1 -11827.8,E2 -11827.8} C_VEL
LIN {X 0,Y 387.481,Z 396.031,A -85,B 0,C 180,E1 -11829.831,E2 -11829.831} C_VEL
LIN {X 0,Y 382.998,Z 383.601,A -85,B 0,C 180,E1 -11832.121,E2 -11832.121} C_VEL
LIN {X 0,Y 382.975,Z 383.386,A -85,B 0,C 180,E1 -11835.786,E2 -11835.786} C_VEL
LIN {X 0,Y 382.964,Z 383.391,A -85,B 0,C 180,E1 -11838.802,E2 -11838.802} C_VEL
LIN {X 0,Y 382.995,Z 383.403,A -85,B 0,C 180,E1 -11842.099,E2 -11842.099} C_VEL
LIN {X 0,Y 383.016,Z 383.37,A -85,B 0,C 180,E1 -11845.332,E2 -11845.332} C_VEL
LIN {X 0,Y 382.983,Z 383.407,A -85,B 0,C 180,E1 -11849.081,E2 -11849.081} C_VEL
LIN {X 0,Y 382.971,Z 383.405,A -85,B 0,C 180,E1 -11852.691,E2 -11852.691} C_VEL
LIN {X 0,Y 383.044,Z 383.639,A -85,B 0,C 180,E1 -11854.158,E2 -11854.158} C_VEL
LIN {X 0,Y 384.32,Z 388.878,A -85,B 0,C 180,E1 -11855.278,E2 -11855.278} C_VEL
LIN {X 0,Y 393.176,Z 412.54,A -85,B 0,C 180,E1 -11856.384,E2 -11856.384} C_VEL
LIN {X 0,Y 389.963,Z 531.829,A -85,B 0,C 180,E1 -11859.18,E2 -11859.18} C_VEL
LIN {X 0,Y 389.568,Z 547.601,A -85,B 0,C 180,E1 -11859.78,E2 -11859.78} C_VEL
LIN {X 0,Y 389.038,Z 562.079,A -85,B 0,C 180,E1 -11860.544,E2 -11860.544} C_VEL
LIN {X 0,Y 388.248,Z 576.489,A -85,B 0,C 180,E1 -11861.531,E2 -11861.531} C_VEL
LIN {X 0,Y 387.533,Z 590.104,A -85,B 0,C 180,E1 -11862.725,E2 -11862.725} C_VEL
LIN {X 0,Y 386.68,Z 602.432,A -85,B 0,C 180,E1 -11864.044,E2 -11864.044} C_VEL
LIN {X 0,Y 385.987,Z 613.642,A -85,B 0,C 180,E1 -11865.501,E2 -11865.501} C_VEL
LIN {X 0,Y 385.146,Z 623.774,A -85,B 0,C 180,E1 -11867.083,E2 -11867.083} C_VEL
LIN {X 0,Y 384.601,Z 632.188,A -85,B 0,C 180,E1 -11868.671,E2 -11868.671} C_VEL
LIN {X 0,Y 384.08,Z 640.25,A -85,B 0,C 180,E1 -11870.521,E2 -11870.521} C_VEL
LIN {X 0,Y 383.792,Z 645.913,A -85,B 0,C 180,E1 -11872.106,E2 -11872.106} C_VEL
LIN {X 0,Y 383.502,Z 650.508,A -85,B 0,C 180,E1 -11873.687,E2 -11873.687} C_VEL
LIN {X 0,Y 383.054,Z 655.301,A -85,B 0,C 180,E1 -11875.791,E2 -11875.791} C_VEL
LIN {X 0,Y 383.202,Z 657.069,A -85,B 0,C 180,E1 -11876.846,E2 -11876.846} C_VEL
LIN {X 0,Y 383.148,Z 659.538,A -85,B 0,C 180,E1 -11878.949,E2 -11878.949} C_VEL
LIN {X 0,Y 383.272,Z 660.59,A -85,B 0,C 180,E1 -11881.051,E2 -11881.051} C_VEL
LIN {X 0,Y 383.623,Z 660.214,A -85,B 0,C 180,E1 -11883.15,E2 -11883.15} C_VEL
LIN {X 0,Y 383.988,Z 658.448,A -85,B 0,C 180,E1 -11885.251,E2 -11885.251} C_VEL
LIN {X 0,Y 384.637,Z 655.213,A -85,B 0,C 180,E1 -11887.348,E2 -11887.348} C_VEL
LIN {X 0,Y 385.321,Z 651.704,A -85,B 0,C 180,E1 -11888.919,E2 -11888.919} C_VEL
LIN {X 0,Y 386.035,Z 647.114,A -85,B 0,C 180,E1 -11890.543,E2 -11890.543} C_VEL
LIN {X 0,Y 387.175,Z 639.742,A -85,B 0,C 180,E1 -11892.581,E2 -11892.581} C_VEL
LIN {X 0,Y 388.182,Z 632.689,A -85,B 0,C 180,E1 -11894.147,E2 -11894.147} C_VEL
LIN {X 0,Y 389.366,Z 624.143,A -85,B 0,C 180,E1 -11895.709,E2 -11895.709} C_VEL
LIN {X 0,Y 390.53,Z 615.54,A -85,B 0,C 180,E1 -11897.012,E2 -11897.012} C_VEL
LIN {X 0,Y 391.798,Z 604.518,A -85,B 0,C 180,E1 -11898.43,E2 -11898.43} C_VEL
LIN {X 0,Y 393.055,Z 592.194,A -85,B 0,C 180,E1 -11899.724,E2 -11899.724} C_VEL
LIN {X 0,Y 394.105,Z 580.015,A -85,B 0,C 180,E1 -11900.758,E2 -11900.758} C_VEL
LIN {X 0,Y 395.215,Z 564.707,A -85,B 0,C 180,E1 -11901.79,E2 -11901.79} C_VEL
LIN {X 0,Y 396.041,Z 550.255,A -85,B 0,C 180,E1 -11902.53,E2 -11902.53} C_VEL
LIN {X 0,Y 396.58,Z 534.151,A -85,B 0,C 180,E1 -11903.119,E2 -11903.119} C_VEL
LIN {X 0,Y 399.488,Z 487.488,A -85,B 0,C 180,E1 -11904.524,E2 -11904.524} C_VEL
LIN {X 0,Y 404.123,Z 427.252,A -85,B 0,C 180,E1 -11906.39,E2 -11906.39} C_VEL
LIN {X 0,Y 398.845,Z 417.92,A -85,B 0,C 180,E1 -11907.563,E2 -11907.563} C_VEL
LIN {X 0,Y 393.93,Z 410.689,A -85,B 0,C 180,E1 -11908.707,E2 -11908.707} C_VEL
LIN {X 0,Y 391.985,Z 407.668,A -85,B 0,C 180,E1 -11909.279,E2 -11909.279} C_VEL
LIN {X 0,Y 390.708,Z 403.392,A -85,B 0,C 180,E1 -11911.443,E2 -11911.443} C_VEL
LIN {X 0,Y 389.434,Z 399.539,A -85,B 0,C 180,E1 -11914.018,E2 -11914.018} C_VEL
LIN {X 0,Y 388.916,Z 397.767,A -85,B 0,C 180,E1 -11915.59,E2 -11915.59} C_VEL
LIN {X 0,Y 388.265,Z 396.204,A -85,B 0,C 180,E1 -11917.983,E2 -11917.983} C_VEL
LIN {X 0,Y 388.241,Z 395.866,A -85,B 0,C 180,E1 -11920.668,E2 -11920.668} C_VEL
LIN {X 0,Y 388.522,Z 396.369,A -85,B 0,C 180,E1 -11922.126,E2 -11922.126} C_VEL
LIN {X 0,Y 389.599,Z 398.399,A -85,B 0,C 180,E1 -11924.71,E2 -11924.71} C_VEL
LIN {X 0,Y 391.216,Z 402.6,A -85,B 0,C 180,E1 -11927.438,E2 -11927.438} C_VEL
LIN {X 0,Y 392.911,Z 406.945,A -85,B 0,C 180,E1 -11929.409,E2 -11929.409} C_VEL
LIN {X 0,Y 394.896,Z 412.97,A -85,B 0,C 180,E1 -11931.543,E2 -11931.543} C_VEL
LIN {X 0,Y 396.792,Z 419.532,A -85,B 0,C 180,E1 -11933.428,E2 -11933.428} C_VEL
LIN {X 0,Y 398.454,Z 426.715,A -85,B 0,C 180,E1 -11935.167,E2 -11935.167} C_VEL
LIN {X 0,Y 398.855,Z 429.099,A -85,B 0,C 180,E1 -11935.676,E2 -11935.676} C_VEL
LIN {X 0,Y 396.215,Z 443.056,A -85,B 0,C 180,E1 -11937.849,E2 -11937.849} C_VEL
LIN {X 0,Y 395.324,Z 448.443,A -85,B 0,C 180,E1 -11938.625,E2 -11938.625} C_VEL
LIN {X 0,Y 397.823,Z 465.115,A -85,B 0,C 180,E1 -11939.647,E2 -11939.647} C_VEL
LIN {X 0,Y 399.859,Z 484.191,A -85,B 0,C 180,E1 -11940.605,E2 -11940.605} C_VEL
LIN {X 0,Y 400.868,Z 502.836,A -85,B 0,C 180,E1 -11941.372,E2 -11941.372} C_VEL
LIN {X 0,Y 396.907,Z 576.865,A -85,B 0,C 180,E1 -11943.334,E2 -11943.334} C_VEL
LIN {X 0,Y 395.362,Z 641.545,A -85,B 0,C 180,E1 -11944.534,E2 -11944.534} C_VEL
LIN {X 0,Y 394.559,Z 657.43,A -85,B 0,C 180,E1 -11945.043,E2 -11945.043} C_VEL
LIN {X 0,Y 393.509,Z 672.474,A -85,B 0,C 180,E1 -11945.745,E2 -11945.745} C_VEL
LIN {X 0,Y 392.27,Z 686.946,A -85,B 0,C 180,E1 -11946.645,E2 -11946.645} C_VEL
LIN {X 0,Y 390.883,Z 700.115,A -85,B 0,C 180,E1 -11947.676,E2 -11947.676} C_VEL
LIN {X 0,Y 389.288,Z 713.487,A -85,B 0,C 180,E1 -11948.971,E2 -11948.971} C_VEL
LIN {X 0,Y 387.804,Z 725.327,A -85,B 0,C 180,E1 -11950.366,E2 -11950.366} C_VEL
LIN {X 0,Y 386.344,Z 736.708,A -85,B 0,C 180,E1 -11951.985,E2 -11951.985} C_VEL
LIN {X 0,Y 384.962,Z 747.425,A -85,B 0,C 180,E1 -11953.833,E2 -11953.833} C_VEL
LIN {X 0,Y 383.858,Z 756.33,A -85,B 0,C 180,E1 -11955.688,E2 -11955.688} C_VEL
LIN {X 0,Y 383.17,Z 762.716,A -85,B 0,C 180,E1 -11957.284,E2 -11957.284} C_VEL
LIN {X 0,Y 382.398,Z 769.768,A -85,B 0,C 180,E1 -11959.408,E2 -11959.408} C_VEL
LIN {X 0,Y 381.996,Z 775.306,A -85,B 0,C 180,E1 -11961.535,E2 -11961.535} C_VEL
LIN {X 0,Y 381.787,Z 779.629,A -85,B 0,C 180,E1 -11963.741,E2 -11963.741} C_VEL
LIN {X 0,Y 381.659,Z 782.417,A -85,B 0,C 180,E1 -11965.774,E2 -11965.774} C_VEL
LIN {X 0,Y 381.617,Z 784.161,A -85,B 0,C 180,E1 -11967.888,E2 -11967.888} C_VEL
LIN {X 0,Y 381.652,Z 784.755,A -85,B 0,C 180,E1 -11969.998,E2 -11969.998} C_VEL
LIN {X 0,Y 381.632,Z 784.157,A -85,B 0,C 180,E1 -11972.109,E2 -11972.109} C_VEL
LIN {X 0,Y 381.66,Z 782.409,A -85,B 0,C 180,E1 -11974.222,E2 -11974.222} C_VEL
LIN {X 0,Y 381.762,Z 779.48,A -85,B 0,C 180,E1 -11976.34,E2 -11976.34} C_VEL
LIN {X 0,Y 381.99,Z 775.301,A -85,B 0,C 180,E1 -11978.462,E2 -11978.462} C_VEL
LIN {X 0,Y 382.391,Z 769.756,A -85,B 0,C 180,E1 -11980.589,E2 -11980.589} C_VEL
LIN {X 0,Y 383.152,Z 762.694,A -85,B 0,C 180,E1 -11982.714,E2 -11982.714} C_VEL
LIN {X 0,Y 383.99,Z 755.123,A -85,B 0,C 180,E1 -11984.574,E2 -11984.574} C_VEL
LIN {X 0,Y 385.106,Z 745.991,A -85,B 0,C 180,E1 -11986.43,E2 -11986.43} C_VEL
LIN {X 0,Y 386.336,Z 736.678,A -85,B 0,C 180,E1 -11988.012,E2 -11988.012} C_VEL
LIN {X 0,Y 387.832,Z 725.01,A -85,B 0,C 180,E1 -11989.668,E2 -11989.668} C_VEL
LIN {X 0,Y 389.404,Z 712.222,A -85,B 0,C 180,E1 -11991.157,E2 -11991.157} C_VEL
LIN {X 0,Y 391.007,Z 698.508,A -85,B 0,C 180,E1 -11992.452,E2 -11992.452} C_VEL
LIN {X 0,Y 392.36,Z 685.102,A -85,B 0,C 180,E1 -11993.477,E2 -11993.477} C_VEL
LIN {X 0,Y 393.563,Z 671.212,A -85,B 0,C 180,E1 -11994.317,E2 -11994.317} C_VEL
LIN {X 0,Y 394.627,Z 655.808,A -85,B 0,C 180,E1 -11995.011,E2 -11995.011} C_VEL
LIN {X 0,Y 395.308,Z 641.31,A -85,B 0,C 180,E1 -11995.467,E2 -11995.467} C_VEL
LIN {X 0,Y 397.499,Z 544.26,A -85,B 0,C 180,E1 -11997.258,E2 -11997.258} C_VEL
LIN {X 0,Y 398.231,Z 500.871,A -85,B 0,C 180,E1 -11998.067,E2 -11998.067} C_VEL
LIN {X 0,Y 394.249,Z 470.073,A -85,B 0,C 180,E1 -11999.002,E2 -11999.002} C_VEL
LIN {X 0,Y 393.556,Z 464.367,A -85,B 0,C 180,E1 -11999.222,E2 -11999.222} C_VEL
LIN {X 0,Y 392.088,Z 444.161,A -85,B 0,C 180,E1 -12000.367,E2 -12000.367} C_VEL
LIN {X 0,Y 394.144,Z 423.129,A -85,B 0,C 180,E1 -12003.064,E2 -12003.064} C_VEL
LIN {X 0,Y 392.803,Z 417.318,A -85,B 0,C 180,E1 -12003.94,E2 -12003.94} C_VEL
LIN {X 0,Y 387.294,Z 398.061,A -85,B 0,C 180,E1 -12007.019,E2 -12007.019} C_VEL
LIN {X 0,Y 382.996,Z 383.654,A -85,B 0,C 180,E1 -12009.48,E2 -12009.48} C_VEL
LIN {X 0,Y 382.95,Z 383.409,A -85,B 0,C 180,E1 -12011.349,E2 -12011.349} C_VEL
LIN {X 0,Y 382.982,Z 383.406,A -85,B 0,C 180,E1 -12014.301,E2 -12014.301} C_VEL
LIN {X 0,Y 382.969,Z 383.37,A -85,B 0,C 180,E1 -12017.235,E2 -12017.235} C_VEL
LIN {X 0,Y 382.972,Z 383.402,A -85,B 0,C 180,E1 -12020.418,E2 -12020.418} C_VEL
LIN {X 0,Y 382.999,Z 383.359,A -85,B 0,C 180,E1 -12024.042,E2 -12024.042} C_VEL
LIN {X 0,Y 382.972,Z 383.399,A -85,B 0,C 180,E1 -12027.577,E2 -12027.577} C_VEL
LIN {X 0,Y 382.963,Z 383.397,A -85,B 0,C 180,E1 -12030.298,E2 -12030.298} C_VEL
LIN {X 0,Y 382.989,Z 383.399,A -85,B 0,C 180,E1 -12034.044,E2 -12034.044} C_VEL
LIN {X 0,Y 382.973,Z 383.404,A -85,B 0,C 180,E1 -12037.333,E2 -12037.333} C_VEL
LIN {X 0,Y 383.027,Z 383.387,A -85,B 0,C 180,E1 -12040.715,E2 -12040.715} C_VEL
LIN {X 0,Y 383.004,Z 383.394,A -85,B 0,C 180,E1 -12044.023,E2 -12044.023} C_VEL
LIN {X 0,Y 383.12,Z 383.385,A -85,B 0,C 180,E1 -12047.283,E2 -12047.283} C_VEL
LIN {X 0,Y 383.122,Z 383.371,A -85,B 0,C 180,E1 -12050.497,E2 -12050.497} C_VEL
LIN {X 0,Y 383.213,Z 383.372,A -85,B 0,C 180,E1 -12053.683,E2 -12053.683} C_VEL
LIN {X 0,Y 383.36,Z 383.353,A -85,B 0,C 180,E1 -12057.899,E2 -12057.899} C_VEL
LIN {X 0,Y 383.357,Z 383.343,A -85,B 0,C 180,E1 -12062.101,E2 -12062.101} C_VEL
LIN {X 0,Y 383.217,Z 383.359,A -85,B 0,C 180,E1 -12066.696,E2 -12066.696} C_VEL
LIN {X 0,Y 383.125,Z 383.383,A -85,B 0,C 180,E1 -12069.503,E2 -12069.503} C_VEL
LIN {X 0,Y 383.111,Z 383.383,A -85,B 0,C 180,E1 -12073.537,E2 -12073.537} C_VEL
LIN {X 0,Y 383.079,Z 383.379,A -85,B 0,C 180,E1 -12077.07,E2 -12077.07} C_VEL
LIN {X 0,Y 383.014,Z 383.389,A -85,B 0,C 180,E1 -12080.648,E2 -12080.648} C_VEL
LIN {X 0,Y 382.995,Z 383.401,A -85,B 0,C 180,E1 -12083.81,E2 -12083.81} C_VEL
LIN {X 0,Y 382.953,Z 383.408,A -85,B 0,C 180,E1 -12087.31,E2 -12087.31} C_VEL
LIN {X 0,Y 382.966,Z 383.411,A -85,B 0,C 180,E1 -12090.92,E2 -12090.92} C_VEL
LIN {X 0,Y 382.999,Z 383.406,A -85,B 0,C 180,E1 -12094.67,E2 -12094.67} C_VEL
LIN {X 0,Y 382.98,Z 383.374,A -85,B 0,C 180,E1 -12097.904,E2 -12097.904} C_VEL
LIN {X 0,Y 382.949,Z 383.395,A -85,B 0,C 180,E1 -12101.352,E2 -12101.352} C_VEL
LIN {X 0,Y 382.977,Z 383.402,A -85,B 0,C 180,E1 -12104.304,E2 -12104.304} C_VEL
LIN {X 0,Y 382.98,Z 383.492,A -85,B 0,C 180,E1 -12107.935,E2 -12107.935} C_VEL
LIN {X 0,Y 383.267,Z 384.768,A -85,B 0,C 180,E1 -12108.236,E2 -12108.236} C_VEL
LIN {X 0,Y 387.758,Z 396.789,A -85,B 0,C 180,E1 -12110.412,E2 -12110.412} C_VEL
LIN {X 0,Y 392.408,Z 411.067,A -85,B 0,C 180,E1 -12112.843,E2 -12112.843} C_VEL
LIN {X 0,Y 396.272,Z 424.938,A -85,B 0,C 180,E1 -12115.073,E2 -12115.073} C_VEL
LIN {X 0,Y 396.901,Z 427.619,A -85,B 0,C 180,E1 -12115.487,E2 -12115.487} C_VEL
LIN {X 0,Y 394.883,Z 454.247,A -85,B 0,C 180,E1 -12118.749,E2 -12118.749} C_VEL
LIN {X 0,Y 393.832,Z 471.629,A -85,B 0,C 180,E1 -12120.754,E2 -12120.754} C_VEL
LIN {X 0,Y 398.93,Z 503.466,A -85,B 0,C 180,E1 -12121.814,E2 -12121.814} C_VEL
LIN {X 0,Y 396.779,Z 608.7,A -85,B 0,C 180,E1 -12123.754,E2 -12123.754} C_VEL
LIN {X 0,Y 395.907,Z 642.277,A -85,B 0,C 180,E1 -12124.399,E2 -12124.399} C_VEL
LIN {X 0,Y 395.151,Z 657.363,A -85,B 0,C 180,E1 -12124.884,E2 -12124.884} C_VEL
LIN {X 0,Y 394.07,Z 671.842,A -85,B 0,C 180,E1 -12125.545,E2 -12125.545} C_VEL
LIN {X 0,Y 392.858,Z 686.015,A -85,B 0,C 180,E1 -12126.407,E2 -12126.407} C_VEL
LIN {X 0,Y 391.379,Z 699.446,A -85,B 0,C 180,E1 -12127.431,E2 -12127.431} C_VEL
LIN {X 0,Y 389.934,Z 711.843,A -85,B 0,C 180,E1 -12128.596,E2 -12128.596} C_VEL
LIN {X 0,Y 388.511,Z 723.366,A -85,B 0,C 180,E1 -12129.899,E2 -12129.899} C_VEL
LIN {X 0,Y 387.009,Z 734.954,A -85,B 0,C 180,E1 -12131.472,E2 -12131.472} C_VEL
LIN {X 0,Y 385.635,Z 744.717,A -85,B 0,C 180,E1 -12133.049,E2 -12133.049} C_VEL
LIN {X 0,Y 384.336,Z 754.267,A -85,B 0,C 180,E1 -12134.898,E2 -12134.898} C_VEL
LIN {X 0,Y 383.443,Z 762.223,A -85,B 0,C 180,E1 -12136.757,E2 -12136.757} C_VEL
LIN {X 0,Y 382.598,Z 769.642,A -85,B 0,C 180,E1 -12138.881,E2 -12138.881} C_VEL
LIN {X 0,Y 382.061,Z 775.646,A -85,B 0,C 180,E1 -12141.055,E2 -12141.055} C_VEL
LIN {X 0,Y 381.799,Z 779.009,A -85,B 0,C 180,E1 -12142.598,E2 -12142.598} C_VEL
LIN {X 0,Y 381.605,Z 782.551,A -85,B 0,C 180,E1 -12144.718,E2 -12144.718} C_VEL
LIN {X 0,Y 381.582,Z 783.519,A -85,B 0,C 180,E1 -12145.497,E2 -12145.497} C_VEL
LIN {X 0,Y 380.924,Z 784.506,A -85,B 0,C 180,E1 -12146.365,E2 -12146.365} C_VEL
LIN {X 0,Y 378.046,Z 785.669,A -85,B 0,C 180,E1 -12147.786,E2 -12147.786} C_VEL
LIN {X 0,Y 375.593,Z 786.149,A -85,B 0,C 180,E1 -12148.941,E2 -12148.941} C_VEL
LIN {X 0,Y 374.527,Z 786.237,A -85,B 0,C 180,E1 -12149.836,E2 -12149.836} C_VEL
LIN {X 0,Y 374.434,Z 786.211,A -85,B 0,C 180,E1 -12150.14,E2 -12150.14} C_VEL
LIN {X 0,Y 374.41,Z 785.661,A -85,B 0,C 180,E1 -12152.153,E2 -12152.153} C_VEL
LIN {X 0,Y 374.499,Z 783.956,A -85,B 0,C 180,E1 -12154.307,E2 -12154.307} C_VEL
LIN {X 0,Y 374.629,Z 781.077,A -85,B 0,C 180,E1 -12156.464,E2 -12156.464} C_VEL
LIN {X 0,Y 374.922,Z 776.957,A -85,B 0,C 180,E1 -12158.626,E2 -12158.626} C_VEL
LIN {X 0,Y 375.356,Z 771.499,A -85,B 0,C 180,E1 -12160.793,E2 -12160.793} C_VEL
LIN {X 0,Y 376.185,Z 764.55,A -85,B 0,C 180,E1 -12162.957,E2 -12162.957} C_VEL
LIN {X 0,Y 377.077,Z 757.102,A -85,B 0,C 180,E1 -12164.851,E2 -12164.851} C_VEL
LIN {X 0,Y 378.328,Z 748.129,A -85,B 0,C 180,E1 -12166.736,E2 -12166.736} C_VEL
LIN {X 0,Y 379.655,Z 738.965,A -85,B 0,C 180,E1 -12168.344,E2 -12168.344} C_VEL
LIN {X 0,Y 381.19,Z 727.866,A -85,B 0,C 180,E1 -12169.984,E2 -12169.984} C_VEL
LIN {X 0,Y 382.724,Z 716.307,A -85,B 0,C 180,E1 -12171.407,E2 -12171.407} C_VEL
LIN {X 0,Y 384.353,Z 703.376,A -85,B 0,C 180,E1 -12172.724,E2 -12172.724} C_VEL
LIN {X 0,Y 385.853,Z 690.804,A -85,B 0,C 180,E1 -12173.767,E2 -12173.767} C_VEL
LIN {X 0,Y 387.191,Z 677.244,A -85,B 0,C 180,E1 -12174.677,E2 -12174.677} C_VEL
LIN {X 0,Y 388.374,Z 661.906,A -85,B 0,C 180,E1 -12175.471,E2 -12175.471} C_VEL
LIN {X 0,Y 389.372,Z 646.439,A -85,B 0,C 180,E1 -12176.031,E2 -12176.031} C_VEL
LIN {X 0,Y 389.918,Z 629.45,A -85,B 0,C 180,E1 -12176.423,E2 -12176.423} C_VEL
LIN {X 0,Y 392.293,Z 526.211,A -85,B 0,C 180,E1 -12178.34,E2 -12178.34} C_VEL
LIN {X 0,Y 392.694,Z 504.268,A -85,B 0,C 180,E1 -12178.757,E2 -12178.757} C_VEL
LIN {X 0,Y 387.442,Z 471.65,A -85,B 0,C 180,E1 -12179.874,E2 -12179.874} C_VEL
LIN {X 0,Y 388.507,Z 455.338,A -85,B 0,C 180,E1 -12181.764,E2 -12181.764} C_VEL
LIN {X 0,Y 390.485,Z 430.46,A -85,B 0,C 180,E1 -12184.852,E2 -12184.852} C_VEL
LIN {X 0,Y 387.593,Z 419.173,A -85,B 0,C 180,E1 -12186.645,E2 -12186.645} C_VEL
LIN {X 0,Y 382.954,Z 403.929,A -85,B 0,C 180,E1 -12189.225,E2 -12189.225} C_VEL
LIN {X 0,Y 378.267,Z 390.831,A -85,B 0,C 180,E1 -12191.598,E2 -12191.598} C_VEL
LIN {X 0,Y 375.965,Z 384.474,A -85,B 0,C 180,E1 -12192.838,E2 -12192.838} C_VEL
LIN {X 0,Y 375.907,Z 384.268,A -85,B 0,C 180,E1 -12196.231,E2 -12196.231} C_VEL
LIN {X 0,Y 375.942,Z 384.255,A -85,B 0,C 180,E1 -12200.04,E2 -12200.04} C_VEL
LIN {X 0,Y 375.961,Z 384.269,A -85,B 0,C 180,E1 -12203.498,E2 -12203.498} C_VEL
LIN {X 0,Y 375.962,Z 384.251,A -85,B 0,C 180,E1 -12205.889,E2 -12205.889} C_VEL
LIN {X 0,Y 375.965,Z 384.28,A -85,B 0,C 180,E1 -12209.687,E2 -12209.687} C_VEL
LIN {X 0,Y 375.921,Z 384.284,A -85,B 0,C 180,E1 -12212.135,E2 -12212.135} C_VEL
LIN {X 0,Y 375.97,Z 384.462,A -85,B 0,C 180,E1 -12213.803,E2 -12213.803} C_VEL
LIN {X 0,Y 377.15,Z 389.369,A -85,B 0,C 180,E1 -12214.874,E2 -12214.874} C_VEL
LIN {X 0,Y 386.422,Z 413.871,A -85,B 0,C 180,E1 -12216.056,E2 -12216.056} C_VEL
LIN {X 0,Y 383.13,Z 531.994,A -85,B 0,C 180,E1 -12218.9,E2 -12218.9} C_VEL
LIN {X 0,Y 382.706,Z 547.724,A -85,B 0,C 180,E1 -12219.503,E2 -12219.503} C_VEL
LIN {X 0,Y 382.158,Z 562.943,A -85,B 0,C 180,E1 -12220.32,E2 -12220.32} C_VEL
LIN {X 0,Y 381.348,Z 577.33,A -85,B 0,C 180,E1 -12221.324,E2 -12221.324} C_VEL
LIN {X 0,Y 380.588,Z 590.951,A -85,B 0,C 180,E1 -12222.538,E2 -12222.538} C_VEL
LIN {X 0,Y 379.715,Z 603.294,A -85,B 0,C 180,E1 -12223.881,E2 -12223.881} C_VEL
LIN {X 0,Y 379.055,Z 613.578,A -85,B 0,C 180,E1 -12225.23,E2 -12225.23} C_VEL
LIN {X 0,Y 378.193,Z 623.908,A -85,B 0,C 180,E1 -12226.842,E2 -12226.842} C_VEL
LIN {X 0,Y 377.64,Z 632.49,A -85,B 0,C 180,E1 -12228.459,E2 -12228.459} C_VEL
LIN {X 0,Y 377.082,Z 640.754,A -85,B 0,C 180,E1 -12230.343,E2 -12230.343} C_VEL
LIN {X 0,Y 376.765,Z 646.504,A -85,B 0,C 180,E1 -12231.958,E2 -12231.958} C_VEL
LIN {X 0,Y 376.487,Z 651.218,A -85,B 0,C 180,E1 -12233.569,E2 -12233.569} C_VEL
LIN {X 0,Y 376.022,Z 656.128,A -85,B 0,C 180,E1 -12235.712,E2 -12235.712} C_VEL
LIN {X 0,Y 376.179,Z 657.965,A -85,B 0,C 180,E1 -12236.787,E2 -12236.787} C_VEL
LIN {X 0,Y 376.125,Z 660.56,A -85,B 0,C 180,E1 -12238.929,E2 -12238.929} C_VEL
LIN {X 0,Y 376.276,Z 661.709,A -85,B 0,C 180,E1 -12241.07,E2 -12241.07} C_VEL
LIN {X 0,Y 376.646,Z 661.434,A -85,B 0,C 180,E1 -12243.209,E2 -12243.209} C_VEL
LIN {X 0,Y 377.04,Z 659.765,A -85,B 0,C 180,E1 -12245.348,E2 -12245.348} C_VEL
LIN {X 0,Y 377.303,Z 658.389,A -85,B 0,C 180,E1 -12246.417,E2 -12246.417} C_VEL
LIN {X 0,Y 378.041,Z 655.554,A -85,B 0,C 180,E1 -12248.015,E2 -12248.015} C_VEL
LIN {X 0,Y 378.631,Z 651.907,A -85,B 0,C 180,E1 -12249.617,E2 -12249.617} C_VEL
LIN {X 0,Y 379.452,Z 647.233,A -85,B 0,C 180,E1 -12251.213,E2 -12251.213} C_VEL
LIN {X 0,Y 380.641,Z 640.429,A -85,B 0,C 180,E1 -12253.072,E2 -12253.072} C_VEL
LIN {X 0,Y 381.949,Z 631.891,A -85,B 0,C 180,E1 -12254.928,E2 -12254.928} C_VEL
LIN {X 0,Y 383.233,Z 622.986,A -85,B 0,C 180,E1 -12256.514,E2 -12256.514} C_VEL
LIN {X 0,Y 384.744,Z 612.128,A -85,B 0,C 180,E1 -12258.091,E2 -12258.091} C_VEL
LIN {X 0,Y 386.056,Z 601.147,A -85,B 0,C 180,E1 -12259.404,E2 -12259.404} C_VEL
LIN {X 0,Y 387.377,Z 587.881,A -85,B 0,C 180,E1 -12260.719,E2 -12260.719} C_VEL
LIN {X 0,Y 388.601,Z 574.485,A -85,B 0,C 180,E1 -12261.762,E2 -12261.762} C_VEL
LIN {X 0,Y 389.569,Z 560.624,A -85,B 0,C 180,E1 -12262.616,E2 -12262.616} C_VEL
LIN {X 0,Y 390.393,Z 544.961,A -85,B 0,C 180,E1 -12263.345,E2 -12263.345} C_VEL
LIN {X 0,Y 391.423,Z 522.907,A -85,B 0,C 180,E1 -12264.073,E2 -12264.073} C_VEL
LIN {X 0,Y 397.06,Z 450.8,A -85,B 0,C 180,E1 -12266.334,E2 -12266.334} C_VEL
LIN {X 0,Y 398.811,Z 430.311,A -85,B 0,C 180,E1 -12266.994,E2 -12266.994} C_VEL
LIN {X 0,Y 394.064,Z 421.983,A -85,B 0,C 180,E1 -12268.117,E2 -12268.117} C_VEL
LIN {X 0,Y 389.972,Z 415.884,A -85,B 0,C 180,E1 -12269.137,E2 -12269.137} C_VEL
LIN {X 0,Y 387.257,Z 412.162,A -85,B 0,C 180,E1 -12269.862,E2 -12269.862} C_VEL
LIN {X 0,Y 385.598,Z 409.582,A -85,B 0,C 180,E1 -12270.428,E2 -12270.428} C_VEL
LIN {X 0,Y 384.174,Z 404.929,A -85,B 0,C 180,E1 -12273.286,E2 -12273.286} C_VEL
LIN {X 0,Y 383.247,Z 401.786,A -85,B 0,C 180,E1 -12276.207,E2 -12276.207} C_VEL
LIN {X 0,Y 382.812,Z 400.624,A -85,B 0,C 180,E1 -12278.623,E2 -12278.623} C_VEL
LIN {X 0,Y 382.975,Z 400.679,A -85,B 0,C 180,E1 -12281.2,E2 -12281.2} C_VEL
LIN {X 0,Y 383.342,Z 401.463,A -85,B 0,C 180,E1 -12282.831,E2 -12282.831} C_VEL
LIN {X 0,Y 384.134,Z 402.867,A -85,B 0,C 180,E1 -12284.475,E2 -12284.475} C_VEL
LIN {X 0,Y 385.433,Z 406.228,A -85,B 0,C 180,E1 -12286.833,E2 -12286.833} C_VEL
LIN {X 0,Y 387.276,Z 411.07,A -85,B 0,C 180,E1 -12289.208,E2 -12289.208} C_VEL
LIN {X 0,Y 389.153,Z 416.893,A -85,B 0,C 180,E1 -12291.344,E2 -12291.344} C_VEL
LIN {X 0,Y 390.909,Z 423.185,A -85,B 0,C 180,E1 -12293.198,E2 -12293.198} C_VEL
LIN {X 0,Y 392.54,Z 430.612,A -85,B 0,C 180,E1 -12295.044,E2 -12295.044} C_VEL
LIN {X 0,Y 392.676,Z 432.357,A -85,B 0,C 180,E1 -12295.416,E2 -12295.416} C_VEL
LIN {X 0,Y 389.74,Z 446.772,A -85,B 0,C 180,E1 -12297.686,E2 -12297.686} C_VEL
LIN {X 0,Y 391.993,Z 462.548,A -85,B 0,C 180,E1 -12298.743,E2 -12298.743} C_VEL
LIN {X 0,Y 393.874,Z 479.3,A -85,B 0,C 180,E1 -12299.674,E2 -12299.674} C_VEL
LIN {X 0,Y 395.024,Z 497.264,A -85,B 0,C 180,E1 -12300.499,E2 -12300.499} C_VEL
LIN {X 0,Y 395.217,Z 504.354,A -85,B 0,C 180,E1 -12300.778,E2 -12300.778} C_VEL
LIN {X 0,Y 390.934,Z 577.685,A -85,B 0,C 180,E1 -12302.786,E2 -12302.786} C_VEL
LIN {X 0,Y 390.162,Z 593.169,A -85,B 0,C 180,E1 -12303.162,E2 -12303.162} C_VEL
LIN {X 0,Y 388.987,Z 641.656,A -85,B 0,C 180,E1 -12304.086,E2 -12304.086} C_VEL
LIN {X 0,Y 388.156,Z 657.413,A -85,B 0,C 180,E1 -12304.598,E2 -12304.598} C_VEL
LIN {X 0,Y 387.038,Z 672.524,A -85,B 0,C 180,E1 -12305.313,E2 -12305.313} C_VEL
LIN {X 0,Y 385.76,Z 687.037,A -85,B 0,C 180,E1 -12306.232,E2 -12306.232} C_VEL
LIN {X 0,Y 384.29,Z 700.149,A -85,B 0,C 180,E1 -12307.272,E2 -12307.272} C_VEL
LIN {X 0,Y 382.626,Z 713.516,A -85,B 0,C 180,E1 -12308.587,E2 -12308.587} C_VEL
LIN {X 0,Y 381.079,Z 725.338,A -85,B 0,C 180,E1 -12310.003,E2 -12310.003} C_VEL
LIN {X 0,Y 379.573,Z 736.731,A -85,B 0,C 180,E1 -12311.652,E2 -12311.652} C_VEL
LIN {X 0,Y 378.292,Z 746.036,A -85,B 0,C 180,E1 -12313.262,E2 -12313.262} C_VEL
LIN {X 0,Y 377.06,Z 755.166,A -85,B 0,C 180,E1 -12315.149,E2 -12315.149} C_VEL
LIN {X 0,Y 376.143,Z 762.734,A -85,B 0,C 180,E1 -12317.042,E2 -12317.042} C_VEL
LIN {X 0,Y 375.569,Z 768.18,A -85,B 0,C 180,E1 -12318.667,E2 -12318.667} C_VEL
LIN {X 0,Y 375.035,Z 774.085,A -85,B 0,C 180,E1 -12320.833,E2 -12320.833} C_VEL
LIN {X 0,Y 374.786,Z 777.575,A -85,B 0,C 180,E1 -12322.456,E2 -12322.456} C_VEL
LIN {X 0,Y 374.618,Z 781.12,A -85,B 0,C 180,E1 -12324.616,E2 -12324.616} C_VEL
LIN {X 0,Y 374.513,Z 783.448,A -85,B 0,C 180,E1 -12326.771,E2 -12326.771} C_VEL
LIN {X 0,Y 374.534,Z 784.617,A -85,B 0,C 180,E1 -12328.923,E2 -12328.923} C_VEL
LIN {X 0,Y 374.535,Z 784.616,A -85,B 0,C 180,E1 -12331.074,E2 -12331.074} C_VEL
LIN {X 0,Y 374.517,Z 783.441,A -85,B 0,C 180,E1 -12333.226,E2 -12333.226} C_VEL
LIN {X 0,Y 374.598,Z 781.109,A -85,B 0,C 180,E1 -12335.381,E2 -12335.381} C_VEL
LIN {X 0,Y 374.782,Z 777.567,A -85,B 0,C 180,E1 -12337.541,E2 -12337.541} C_VEL
LIN {X 0,Y 375.116,Z 772.722,A -85,B 0,C 180,E1 -12339.706,E2 -12339.706} C_VEL
LIN {X 0,Y 375.785,Z 766.441,A -85,B 0,C 180,E1 -12341.87,E2 -12341.87} C_VEL
LIN {X 0,Y 376.583,Z 758.546,A -85,B 0,C 180,E1 -12344.039,E2 -12344.039} C_VEL
LIN {X 0,Y 377.706,Z 750.114,A -85,B 0,C 180,E1 -12345.928,E2 -12345.928} C_VEL
LIN {X 0,Y 379.031,Z 739.937,A -85,B 0,C 180,E1 -12347.813,E2 -12347.813} C_VEL
LIN {X 0,Y 380.509,Z 729.506,A -85,B 0,C 180,E1 -12349.416,E2 -12349.416} C_VEL
LIN {X 0,Y 382.028,Z 718.14,A -85,B 0,C 180,E1 -12350.879,E2 -12350.879} C_VEL
LIN {X 0,Y 383.573,Z 705.754,A -85,B 0,C 180,E1 -12352.202,E2 -12352.202} C_VEL
LIN {X 0,Y 385.15,Z 692.152,A -85,B 0,C 180,E1 -12353.381,E2 -12353.381} C_VEL
LIN {X 0,Y 386.556,Z 677.967,A -85,B 0,C 180,E1 -12354.362,E2 -12354.362} C_VEL
LIN {X 0,Y 387.657,Z 664.408,A -85,B 0,C 180,E1 -12355.092,E2 -12355.092} C_VEL
LIN {X 0,Y 388.606,Z 648.811,A -85,B 0,C 180,E1 -12355.703,E2 -12355.703} C_VEL
LIN {X 0,Y 389.168,Z 634.026,A -85,B 0,C 180,E1 -12356.078,E2 -12356.078} C_VEL
LIN {X 0,Y 392.055,Z 504.823,A -85,B 0,C 180,E1 -12358.471,E2 -12358.471} C_VEL
LIN {X 0,Y 391.405,Z 496.266,A -85,B 0,C 180,E1 -12358.698,E2 -12358.698} C_VEL
LIN {X 0,Y 387.281,Z 465.149,A -85,B 0,C 180,E1 -12359.713,E2 -12359.713} C_VEL
LIN {X 0,Y 385.598,Z 441.757,A -85,B 0,C 180,E1 -12361.06,E2 -12361.06} C_VEL
LIN {X 0,Y 387.271,Z 423.776,A -85,B 0,C 180,E1 -12363.407,E2 -12363.407} C_VEL
LIN {X 0,Y 382.587,Z 407.072,A -85,B 0,C 180,E1 -12366.073,E2 -12366.073} C_VEL
LIN {X 0,Y 377.219,Z 388.834,A -85,B 0,C 180,E1 -12369.152,E2 -12369.152} C_VEL
LIN {X 0,Y 375.947,Z 384.446,A -85,B 0,C 180,E1 -12369.963,E2 -12369.963} C_VEL
LIN {X 0,Y 375.917,Z 384.286,A -85,B 0,C 180,E1 -12373.765,E2 -12373.765} C_VEL
LIN {X 0,Y 375.92,Z 384.252,A -85,B 0,C 180,E1 -12376.81,E2 -12376.81} C_VEL
LIN {X 0,Y 375.921,Z 384.282,A -85,B 0,C 180,E1 -12380.532,E2 -12380.532} C_VEL
LIN {X 0,Y 375.944,Z 384.244,A -85,B 0,C 180,E1 -12383.496,E2 -12383.496} C_VEL
LIN {X 0,Y 375.944,Z 384.242,A -85,B 0,C 180,E1 -12385.887,E2 -12385.887} C_VEL
LIN {X 0,Y 375.948,Z 384.277,A -85,B 0,C 180,E1 -12389.686,E2 -12389.686} C_VEL
LIN {X 0,Y 375.911,Z 384.28,A -85,B 0,C 180,E1 -12392.135,E2 -12392.135} C_VEL
LIN {X 0,Y 375.921,Z 384.272,A -85,B 0,C 180,E1 -12394.533,E2 -12394.533} C_VEL
LIN {X 0,Y 375.959,Z 384.279,A -85,B 0,C 180,E1 -12396.886,E2 -12396.886} C_VEL
LIN {X 0,Y 375.97,Z 384.263,A -85,B 0,C 180,E1 -12400.338,E2 -12400.338} C_VEL
LIN {X 0,Y 375.96,Z 384.276,A -85,B 0,C 180,E1 -12403.716,E2 -12403.716} C_VEL
LIN {X 0,Y 376.088,Z 384.262,A -85,B 0,C 180,E1 -12407.042,E2 -12407.042} C_VEL
LIN {X 0,Y 376.093,Z 384.246,A -85,B 0,C 180,E1 -12410.318,E2 -12410.318} C_VEL
LIN {X 0,Y 376.173,Z 384.249,A -85,B 0,C 180,E1 -12413.564,E2 -12413.564} C_VEL
LIN {X 0,Y 376.325,Z 384.229,A -85,B 0,C 180,E1 -12417.86,E2 -12417.86} C_VEL
LIN {X 0,Y 376.322,Z 384.22,A -85,B 0,C 180,E1 -12422.141,E2 -12422.141} C_VEL
LIN {X 0,Y 376.181,Z 384.235,A -85,B 0,C 180,E1 -12426.685,E2 -12426.685} C_VEL
LIN {X 0,Y 376.095,Z 384.259,A -85,B 0,C 180,E1 -12429.682,E2 -12429.682} C_VEL
LIN {X 0,Y 376.075,Z 384.26,A -85,B 0,C 180,E1 -12433.658,E2 -12433.658} C_VEL
LIN {X 0,Y 376.018,Z 384.261,A -85,B 0,C 180,E1 -12437.401,E2 -12437.401} C_VEL
LIN {X 0,Y 375.965,Z 384.265,A -85,B 0,C 180,E1 -12440.833,E2 -12440.833} C_VEL
LIN {X 0,Y 375.944,Z 384.278,A -85,B 0,C 180,E1 -12444.285,E2 -12444.285} C_VEL
LIN {X 0,Y 375.902,Z 384.285,A -85,B 0,C 180,E1 -12447.866,E2 -12447.866} C_VEL
LIN {X 0,Y 375.924,Z 384.284,A -85,B 0,C 180,E1 -12450.69,E2 -12450.69} C_VEL
LIN {X 0,Y 375.945,Z 384.283,A -85,B 0,C 180,E1 -12454.113,E2 -12454.113} C_VEL
LIN {X 0,Y 375.936,Z 384.253,A -85,B 0,C 180,E1 -12456.743,E2 -12456.743} C_VEL
LIN {X 0,Y 375.926,Z 384.284,A -85,B 0,C 180,E1 -12459.963,E2 -12459.963} C_VEL
LIN {X 0,Y 375.913,Z 384.269,A -85,B 0,C 180,E1 -12463.769,E2 -12463.769} C_VEL
LIN {X 0,Y 375.96,Z 384.338,A -85,B 0,C 180,E1 -12467.211,E2 -12467.211} C_VEL
LIN {X 0,Y 376.049,Z 384.899,A -85,B 0,C 180,E1 -12467.399,E2 -12467.399} C_VEL
LIN {X 0,Y 381.554,Z 399.819,A -85,B 0,C 180,E1 -12470.152,E2 -12470.152} C_VEL
LIN {X 0,Y 386.629,Z 415.616,A -85,B 0,C 180,E1 -12472.88,E2 -12472.88} C_VEL
LIN {X 0,Y 390.394,Z 429.578,A -85,B 0,C 180,E1 -12475.143,E2 -12475.143} C_VEL
LIN {X 0,Y 388.542,Z 454.442,A -85,B 0,C 180,E1 -12478.227,E2 -12478.227} C_VEL
LIN {X 0,Y 387.378,Z 471.279,A -85,B 0,C 180,E1 -12480.2,E2 -12480.2} C_VEL
LIN {X 0,Y 392.543,Z 503.516,A -85,B 0,C 180,E1 -12481.317,E2 -12481.317} C_VEL
LIN {X 0,Y 392.698,Z 508.189,A -85,B 0,C 180,E1 -12481.425,E2 -12481.425} C_VEL
LIN {X 0,Y 389.625,Z 639.471,A -85,B 0,C 180,E1 -12483.883,E2 -12483.883} C_VEL
LIN {X 0,Y 388.853,Z 655.187,A -85,B 0,C 180,E1 -12484.359,E2 -12484.359} C_VEL
LIN {X 0,Y 387.736,Z 670.302,A -85,B 0,C 180,E1 -12485.032,E2 -12485.032} C_VEL
LIN {X 0,Y 386.514,Z 684.062,A -85,B 0,C 180,E1 -12485.853,E2 -12485.853} C_VEL
LIN {X 0,Y 385.019,Z 697.879,A -85,B 0,C 180,E1 -12486.895,E2 -12486.895} C_VEL
LIN {X 0,Y 383.463,Z 710.558,A -85,B 0,C 180,E1 -12488.075,E2 -12488.075} C_VEL
LIN {X 0,Y 381.938,Z 722.298,A -85,B 0,C 180,E1 -12489.397,E2 -12489.397} C_VEL
LIN {X 0,Y 380.448,Z 733.183,A -85,B 0,C 180,E1 -12490.861,E2 -12490.861} C_VEL
LIN {X 0,Y 379.002,Z 743.22,A -85,B 0,C 180,E1 -12492.464,E2 -12492.464} C_VEL
LIN {X 0,Y 377.649,Z 753.026,A -85,B 0,C 180,E1 -12494.347,E2 -12494.347} C_VEL
LIN {X 0,Y 376.599,Z 761.049,A -85,B 0,C 180,E1 -12496.208,E2 -12496.208} C_VEL
LIN {X 0,Y 375.822,Z 767.909,A -85,B 0,C 180,E1 -12498.131,E2 -12498.131} C_VEL
LIN {X 0,Y 375.121,Z 774.162,A -85,B 0,C 180,E1 -12500.294,E2 -12500.294} C_VEL
LIN {X 0,Y 374.719,Z 778.995,A -85,B 0,C 180,E1 -12502.458,E2 -12502.458} C_VEL
LIN {X 0,Y 374.518,Z 782.537,A -85,B 0,C 180,E1 -12504.618,E2 -12504.618} C_VEL
LIN {X 0,Y 374.421,Z 784.879,A -85,B 0,C 180,E1 -12506.774,E2 -12506.774} C_VEL
LIN {X 0,Y 374.449,Z 786.071,A -85,B 0,C 180,E1 -12508.926,E2 -12508.926} C_VEL
LIN {X 0,Y 374.434,Z 786.211,A -85,B 0,C 180,E1 -12510.14,E2 -12510.14} C_VEL
LIN {X 0,Y 373.748,Z 786.091,A -85,B 0,C 180,E1 -12511.037,E2 -12511.037} C_VEL
LIN {X 0,Y 370.889,Z 785.5,A -85,B 0,C 180,E1 -12512.496,E2 -12512.496} C_VEL
LIN {X 0,Y 368.492,Z 784.654,A -85,B 0,C 180,E1 -12513.67,E2 -12513.67} C_VEL
LIN {X 0,Y 367.483,Z 783.756,A -85,B 0,C 180,E1 -12514.572,E2 -12514.572} C_VEL
LIN {X 0,Y 367.41,Z 783.37,A -85,B 0,C 180,E1 -12514.877,E2 -12514.877} C_VEL
LIN {X 0,Y 367.557,Z 781.062,A -85,B 0,C 180,E1 -12516.589,E2 -12516.589} C_VEL
LIN {X 0,Y 367.849,Z 776.941,A -85,B 0,C 180,E1 -12518.793,E2 -12518.793} C_VEL
LIN {X 0,Y 368.333,Z 771.482,A -85,B 0,C 180,E1 -12521.001,E2 -12521.001} C_VEL
LIN {X 0,Y 369.208,Z 764.531,A -85,B 0,C 180,E1 -12523.206,E2 -12523.206} C_VEL
LIN {X 0,Y 370.168,Z 757.082,A -85,B 0,C 180,E1 -12525.134,E2 -12525.134} C_VEL
LIN {X 0,Y 371.474,Z 748.108,A -85,B 0,C 180,E1 -12527.054,E2 -12527.054} C_VEL
LIN {X 0,Y 372.877,Z 738.942,A -85,B 0,C 180,E1 -12528.69,E2 -12528.69} C_VEL
LIN {X 0,Y 374.608,Z 726.875,A -85,B 0,C 180,E1 -12530.494,E2 -12530.494} C_VEL
LIN {X 0,Y 376.285,Z 715.127,A -85,B 0,C 180,E1 -12531.936,E2 -12531.936} C_VEL
LIN {X 0,Y 377.972,Z 701.947,A -85,B 0,C 180,E1 -12533.275,E2 -12533.275} C_VEL
LIN {X 0,Y 379.574,Z 689.048,A -85,B 0,C 180,E1 -12534.33,E2 -12534.33} C_VEL
LIN {X 0,Y 380.962,Z 674.592,A -85,B 0,C 180,E1 -12535.282,E2 -12535.282} C_VEL
LIN {X 0,Y 382.189,Z 659.546,A -85,B 0,C 180,E1 -12536.029,E2 -12536.029} C_VEL
LIN {X 0,Y 383.142,Z 644.228,A -85,B 0,C 180,E1 -12536.56,E2 -12536.56} C_VEL
LIN {X 0,Y 383.701,Z 623.942,A -85,B 0,C 180,E1 -12536.996,E2 -12536.996} C_VEL
LIN {X 0,Y 386.05,Z 526.268,A -85,B 0,C 180,E1 -12538.837,E2 -12538.837} C_VEL
LIN {X 0,Y 386.464,Z 505.239,A -85,B 0,C 180,E1 -12539.242,E2 -12539.242} C_VEL
LIN {X 0,Y 381.078,Z 471.412,A -85,B 0,C 180,E1 -12540.434,E2 -12540.434} C_VEL
LIN {X 0,Y 382.381,Z 452.539,A -85,B 0,C 180,E1 -12542.678,E2 -12542.678} C_VEL
LIN {X 0,Y 384.056,Z 432.472,A -85,B 0,C 180,E1 -12545.201,E2 -12545.201} C_VEL
LIN {X 0,Y 380.076,Z 417.773,A -85,B 0,C 180,E1 -12547.606,E2 -12547.606} C_VEL
LIN {X 0,Y 375.887,Z 404.408,A -85,B 0,C 180,E1 -12549.952,E2 -12549.952} C_VEL
LIN {X 0,Y 371.117,Z 391.272,A -85,B 0,C 180,E1 -12552.391,E2 -12552.391} C_VEL
LIN {X 0,Y 368.875,Z 385.382,A -85,B 0,C 180,E1 -12553.588,E2 -12553.588} C_VEL
LIN {X 0,Y 368.862,Z 385.15,A -85,B 0,C 180,E1 -12556.692,E2 -12556.692} C_VEL
LIN {X 0,Y 368.889,Z 385.134,A -85,B 0,C 180,E1 -12559.649,E2 -12559.649} C_VEL
LIN {X 0,Y 368.9,Z 385.154,A -85,B 0,C 180,E1 -12563.146,E2 -12563.146} C_VEL
LIN {X 0,Y 368.9,Z 385.137,A -85,B 0,C 180,E1 -12566.462,E2 -12566.462} C_VEL
LIN {X 0,Y 368.897,Z 385.16,A -85,B 0,C 180,E1 -12570.308,E2 -12570.308} C_VEL
LIN {X 0,Y 368.919,Z 385.353,A -85,B 0,C 180,E1 -12573.459,E2 -12573.459} C_VEL
LIN {X 0,Y 370.069,Z 390.034,A -85,B 0,C 180,E1 -12574.485,E2 -12574.485} C_VEL
LIN {X 0,Y 379.677,Z 415.375,A -85,B 0,C 180,E1 -12575.732,E2 -12575.732} C_VEL
LIN {X 0,Y 376.737,Z 511.631,A -85,B 0,C 180,E1 -12578.093,E2 -12578.093} C_VEL
LIN {X 0,Y 376.182,Z 535.782,A -85,B 0,C 180,E1 -12578.743,E2 -12578.743} C_VEL
LIN {X 0,Y 375.784,Z 551.29,A -85,B 0,C 180,E1 -12579.39,E2 -12579.39} C_VEL
LIN {X 0,Y 375.19,Z 565.011,A -85,B 0,C 180,E1 -12580.166,E2 -12580.166} C_VEL
LIN {X 0,Y 374.357,Z 579.737,A -85,B 0,C 180,E1 -12581.246,E2 -12581.246} C_VEL
LIN {X 0,Y 373.573,Z 593.117,A -85,B 0,C 180,E1 -12582.482,E2 -12582.482} C_VEL
LIN {X 0,Y 372.685,Z 605.104,A -85,B 0,C 180,E1 -12583.827,E2 -12583.827} C_VEL
LIN {X 0,Y 372.023,Z 615.434,A -85,B 0,C 180,E1 -12585.224,E2 -12585.224} C_VEL
LIN {X 0,Y 371.128,Z 625.651,A -85,B 0,C 180,E1 -12586.865,E2 -12586.865} C_VEL
LIN {X 0,Y 370.591,Z 634.137,A -85,B 0,C 180,E1 -12588.514,E2 -12588.514} C_VEL
LIN {X 0,Y 370.016,Z 642.367,A -85,B 0,C 180,E1 -12590.461,E2 -12590.461} C_VEL
LIN {X 0,Y 369.663,Z 648.815,A -85,B 0,C 180,E1 -12592.352,E2 -12592.352} C_VEL
LIN {X 0,Y 369.368,Z 653.365,A -85,B 0,C 180,E1 -12593.993,E2 -12593.993} C_VEL
LIN {X 0,Y 368.99,Z 656.943,A -85,B 0,C 180,E1 -12595.63,E2 -12595.63} C_VEL
LIN {X 0,Y 369.155,Z 658.83,A -85,B 0,C 180,E1 -12596.726,E2 -12596.726} C_VEL
LIN {X 0,Y 369.101,Z 661.567,A -85,B 0,C 180,E1 -12598.909,E2 -12598.909} C_VEL
LIN {X 0,Y 369.277,Z 662.834,A -85,B 0,C 180,E1 -12601.09,E2 -12601.09} C_VEL
LIN {X 0,Y 369.691,Z 662.654,A -85,B 0,C 180,E1 -12603.269,E2 -12603.269} C_VEL
LIN {X 0,Y 370.093,Z 661.083,A -85,B 0,C 180,E1 -12605.448,E2 -12605.448} C_VEL
LIN {X 0,Y 370.881,Z 658.04,A -85,B 0,C 180,E1 -12607.622,E2 -12607.622} C_VEL
LIN {X 0,Y 371.805,Z 653.473,A -85,B 0,C 180,E1 -12609.795,E2 -12609.795} C_VEL
LIN {X 0,Y 372.816,Z 648.324,A -85,B 0,C 180,E1 -12611.596,E2 -12611.596} C_VEL
LIN {X 0,Y 374.164,Z 641.121,A -85,B 0,C 180,E1 -12613.579,E2 -12613.579} C_VEL
LIN {X 0,Y 375.37,Z 633.896,A -85,B 0,C 180,E1 -12615.196,E2 -12615.196} C_VEL
LIN {X 0,Y 376.744,Z 625.133,A -85,B 0,C 180,E1 -12616.807,E2 -12616.807} C_VEL
LIN {X 0,Y 378.324,Z 614.463,A -85,B 0,C 180,E1 -12618.409,E2 -12618.409} C_VEL
LIN {X 0,Y 379.879,Z 602.661,A -85,B 0,C 180,E1 -12619.874,E2 -12619.874} C_VEL
LIN {X 0,Y 381.294,Z 589.479,A -85,B 0,C 180,E1 -12621.206,E2 -12621.206} C_VEL
LIN {X 0,Y 382.765,Z 574.387,A -85,B 0,C 180,E1 -12622.395,E2 -12622.395} C_VEL
LIN {X 0,Y 383.825,Z 560.636,A -85,B 0,C 180,E1 -12623.248,E2 -12623.248} C_VEL
LIN {X 0,Y 384.625,Z 545.9,A -85,B 0,C 180,E1 -12623.939,E2 -12623.939} C_VEL
LIN {X 0,Y 386.033,Z 519.858,A -85,B 0,C 180,E1 -12624.826,E2 -12624.826} C_VEL
LIN {X 0,Y 393.078,Z 438.997,A -85,B 0,C 180,E1 -12627.452,E2 -12627.452} C_VEL
LIN {X 0,Y 393.607,Z 433.362,A -85,B 0,C 180,E1 -12627.639,E2 -12627.639} C_VEL
LIN {X 0,Y 388.816,Z 425.082,A -85,B 0,C 180,E1 -12628.86,E2 -12628.86} C_VEL
LIN {X 0,Y 384.33,Z 418.507,A -85,B 0,C 180,E1 -12630.078,E2 -12630.078} C_VEL
LIN {X 0,Y 381.127,Z 414.368,A -85,B 0,C 180,E1 -12631.018,E2 -12631.018} C_VEL
LIN {X 0,Y 379.297,Z 411.722,A -85,B 0,C 180,E1 -12631.7,E2 -12631.7} C_VEL
LIN {X 0,Y 378.365,Z 408.643,A -85,B 0,C 180,E1 -12633.865,E2 -12633.865} C_VEL
LIN {X 0,Y 377.689,Z 406.12,A -85,B 0,C 180,E1 -12636.545,E2 -12636.545} C_VEL
LIN {X 0,Y 377.401,Z 405.122,A -85,B 0,C 180,E1 -12639.283,E2 -12639.283} C_VEL
LIN {X 0,Y 377.738,Z 405.649,A -85,B 0,C 180,E1 -12641.906,E2 -12641.906} C_VEL
LIN {X 0,Y 378.331,Z 406.743,A -85,B 0,C 180,E1 -12643.573,E2 -12643.573} C_VEL
LIN {X 0,Y 379.151,Z 408.443,A -85,B 0,C 180,E1 -12645.22,E2 -12645.22} C_VEL
LIN {X 0,Y 380.601,Z 412.305,A -85,B 0,C 180,E1 -12647.614,E2 -12647.614} C_VEL
LIN {X 0,Y 381.97,Z 416.212,A -85,B 0,C 180,E1 -12649.4,E2 -12649.4} C_VEL
LIN {X 0,Y 383.288,Z 420.319,A -85,B 0,C 180,E1 -12650.937,E2 -12650.937} C_VEL
LIN {X 0,Y 385.032,Z 426.842,A -85,B 0,C 180,E1 -12652.96,E2 -12652.96} C_VEL
LIN {X 0,Y 386.398,Z 433.331,A -85,B 0,C 180,E1 -12654.642,E2 -12654.642} C_VEL
LIN {X 0,Y 386.572,Z 435.391,A -85,B 0,C 180,E1 -12655.091,E2 -12655.091} C_VEL
LIN {X 0,Y 384.342,Z 445.577,A -85,B 0,C 180,E1 -12656.729,E2 -12656.729} C_VEL
LIN {X 0,Y 386.724,Z 462.949,A -85,B 0,C 180,E1 -12657.965,E2 -12657.965} C_VEL
LIN {X 0,Y 388.481,Z 479.176,A -85,B 0,C 180,E1 -12658.925,E2 -12658.925} C_VEL
LIN {X 0,Y 389.475,Z 495.165,A -85,B 0,C 180,E1 -12659.711,E2 -12659.711} C_VEL
LIN {X 0,Y 389.71,Z 505.153,A -85,B 0,C 180,E1 -12660.132,E2 -12660.132} C_VEL
LIN {X 0,Y 385.255,Z 575.687,A -85,B 0,C 180,E1 -12662.129,E2 -12662.129} C_VEL
LIN {X 0,Y 383.545,Z 605.882,A -85,B 0,C 180,E1 -12662.919,E2 -12662.919} C_VEL
LIN {X 0,Y 382.611,Z 641.764,A -85,B 0,C 180,E1 -12663.621,E2 -12663.621} C_VEL
LIN {X 0,Y 381.757,Z 657.479,A -85,B 0,C 180,E1 -12664.141,E2 -12664.141} C_VEL
LIN {X 0,Y 380.589,Z 672.574,A -85,B 0,C 180,E1 -12664.866,E2 -12664.866} C_VEL
LIN {X 0,Y 379.266,Z 687.179,A -85,B 0,C 180,E1 -12665.807,E2 -12665.807} C_VEL
LIN {X 0,Y 377.724,Z 700.182,A -85,B 0,C 180,E1 -12666.854,E2 -12666.854} C_VEL
LIN {X 0,Y 376.016,Z 713.544,A -85,B 0,C 180,E1 -12668.192,E2 -12668.192} C_VEL
LIN {X 0,Y 374.328,Z 725.691,A -85,B 0,C 180,E1 -12669.675,E2 -12669.675} C_VEL
LIN {X 0,Y 372.813,Z 736.753,A -85,B 0,C 180,E1 -12671.307,E2 -12671.307} C_VEL
LIN {X 0,Y 371.447,Z 746.057,A -85,B 0,C 180,E1 -12672.945,E2 -12672.945} C_VEL
LIN {X 0,Y 370.153,Z 755.185,A -85,B 0,C 180,E1 -12674.865,E2 -12674.865} C_VEL
LIN {X 0,Y 369.154,Z 762.752,A -85,B 0,C 180,E1 -12676.792,E2 -12676.792} C_VEL
LIN {X 0,Y 368.566,Z 768.197,A -85,B 0,C 180,E1 -12678.449,E2 -12678.449} C_VEL
LIN {X 0,Y 367.972,Z 774.101,A -85,B 0,C 180,E1 -12680.655,E2 -12680.655} C_VEL
LIN {X 0,Y 367.707,Z 777.59,A -85,B 0,C 180,E1 -12682.31,E2 -12682.31} C_VEL
LIN {X 0,Y 367.532,Z 781.134,A -85,B 0,C 180,E1 -12684.512,E2 -12684.512} C_VEL
LIN {X 0,Y 367.428,Z 783.463,A -85,B 0,C 180,E1 -12686.709,E2 -12686.709} C_VEL
LIN {X 0,Y 367.432,Z 784.631,A -85,B 0,C 180,E1 -12688.902,E2 -12688.902} C_VEL
LIN {X 0,Y 367.434,Z 784.629,A -85,B 0,C 180,E1 -12691.094,E2 -12691.094} C_VEL
LIN {X 0,Y 367.431,Z 783.455,A -85,B 0,C 180,E1 -12693.288,E2 -12693.288} C_VEL
LIN {X 0,Y 367.513,Z 781.123,A -85,B 0,C 180,E1 -12695.485,E2 -12695.485} C_VEL
LIN {X 0,Y 367.703,Z 777.581,A -85,B 0,C 180,E1 -12697.687,E2 -12697.687} C_VEL
LIN {X 0,Y 368.078,Z 772.736,A -85,B 0,C 180,E1 -12699.893,E2 -12699.893} C_VEL
LIN {X 0,Y 368.782,Z 766.456,A -85,B 0,C 180,E1 -12702.099,E2 -12702.099} C_VEL
LIN {X 0,Y 369.669,Z 758.561,A -85,B 0,C 180,E1 -12704.307,E2 -12704.307} C_VEL
LIN {X 0,Y 370.831,Z 750.13,A -85,B 0,C 180,E1 -12706.231,E2 -12706.231} C_VEL
LIN {X 0,Y 372.234,Z 739.954,A -85,B 0,C 180,E1 -12708.149,E2 -12708.149} C_VEL
LIN {X 0,Y 373.76,Z 729.525,A -85,B 0,C 180,E1 -12709.781,E2 -12709.781} C_VEL
LIN {X 0,Y 375.34,Z 718.161,A -85,B 0,C 180,E1 -12711.269,E2 -12711.269} C_VEL
LIN {X 0,Y 376.965,Z 705.778,A -85,B 0,C 180,E1 -12712.612,E2 -12712.612} C_VEL
LIN {X 0,Y 378.632,Z 692.18,A -85,B 0,C 180,E1 -12713.808,E2 -12713.808} C_VEL
LIN {X 0,Y 380.051,Z 678.505,A -85,B 0,C 180,E1 -12714.774,E2 -12714.774} C_VEL
LIN {X 0,Y 381.247,Z 664.452,A -85,B 0,C 180,E1 -12715.544,E2 -12715.544} C_VEL
LIN {X 0,Y 382.209,Z 649.453,A -85,B 0,C 180,E1 -12716.145,E2 -12716.145} C_VEL
LIN {X 0,Y 382.825,Z 634.133,A -85,B 0,C 180,E1 -12716.543,E2 -12716.543} C_VEL
LIN {X 0,Y 385.754,Z 508.308,A -85,B 0,C 180,E1 -12718.91,E2 -12718.91} C_VEL
LIN {X 0,Y 385.578,Z 500.859,A -85,B 0,C 180,E1 -12719.079,E2 -12719.079} C_VEL
LIN {X 0,Y 381.251,Z 467.615,A -85,B 0,C 180,E1 -12720.149,E2 -12720.149} C_VEL
LIN {X 0,Y 380.502,Z 458.09,A -85,B 0,C 180,E1 -12720.677,E2 -12720.677} C_VEL
LIN {X 0,Y 379.187,Z 438.96,A -85,B 0,C 180,E1 -12721.813,E2 -12721.813} C_VEL
LIN {X 0,Y 380.497,Z 426.597,A -85,B 0,C 180,E1 -12723.449,E2 -12723.449} C_VEL
LIN {X 0,Y 379.842,Z 423.166,A -85,B 0,C 180,E1 -12723.974,E2 -12723.974} C_VEL
LIN {X 0,Y 374.235,Z 403.383,A -85,B 0,C 180,E1 -12727.226,E2 -12727.226} C_VEL
LIN {X 0,Y 368.898,Z 385.36,A -85,B 0,C 180,E1 -12730.414,E2 -12730.414} C_VEL
LIN {X 0,Y 368.87,Z 385.163,A -85,B 0,C 180,E1 -12733.614,E2 -12733.614} C_VEL
LIN {X 0,Y 368.87,Z 385.13,A -85,B 0,C 180,E1 -12736.694,E2 -12736.694} C_VEL
LIN {X 0,Y 368.872,Z 385.145,A -85,B 0,C 180,E1 -12739.647,E2 -12739.647} C_VEL
LIN {X 0,Y 368.882,Z 385.129,A -85,B 0,C 180,E1 -12743.145,E2 -12743.145} C_VEL
LIN {X 0,Y 368.881,Z 385.132,A -85,B 0,C 180,E1 -12746.461,E2 -12746.461} C_VEL
LIN {X 0,Y 368.899,Z 385.157,A -85,B 0,C 180,E1 -12749.044,E2 -12749.044} C_VEL
LIN {X 0,Y 368.896,Z 385.15,A -85,B 0,C 180,E1 -12751.557,E2 -12751.557} C_VEL
LIN {X 0,Y 368.872,Z 385.145,A -85,B 0,C 180,E1 -12755.219,E2 -12755.219} C_VEL
LIN {X 0,Y 368.884,Z 385.159,A -85,B 0,C 180,E1 -12757.602,E2 -12757.602} C_VEL
LIN {X 0,Y 368.906,Z 385.15,A -85,B 0,C 180,E1 -12761.103,E2 -12761.103} C_VEL
LIN {X 0,Y 368.924,Z 385.14,A -85,B 0,C 180,E1 -12764.532,E2 -12764.532} C_VEL
LIN {X 0,Y 369.042,Z 385.137,A -85,B 0,C 180,E1 -12766.79,E2 -12766.79} C_VEL
LIN {X 0,Y 369.044,Z 385.124,A -85,B 0,C 180,E1 -12770.131,E2 -12770.131} C_VEL
LIN {X 0,Y 369.136,Z 385.126,A -85,B 0,C 180,E1 -12773.441,E2 -12773.441} C_VEL
LIN {X 0,Y 369.289,Z 385.106,A -85,B 0,C 180,E1 -12777.819,E2 -12777.819} C_VEL
LIN {X 0,Y 369.286,Z 385.096,A -85,B 0,C 180,E1 -12782.181,E2 -12782.181} C_VEL
LIN {X 0,Y 369.152,Z 385.11,A -85,B 0,C 180,E1 -12786.671,E2 -12786.671} C_VEL
LIN {X 0,Y 369.046,Z 385.137,A -85,B 0,C 180,E1 -12789.869,E2 -12789.869} C_VEL
LIN {X 0,Y 369.023,Z 385.138,A -85,B 0,C 180,E1 -12793.773,E2 -12793.773} C_VEL
LIN {X 0,Y 368.977,Z 385.141,A -85,B 0,C 180,E1 -12797.744,E2 -12797.744} C_VEL
LIN {X 0,Y 368.895,Z 385.145,A -85,B 0,C 180,E1 -12801.222,E2 -12801.222} C_VEL
LIN {X 0,Y 368.904,Z 385.157,A -85,B 0,C 180,E1 -12803.878,E2 -12803.878} C_VEL
LIN {X 0,Y 368.843,Z 385.167,A -85,B 0,C 180,E1 -12807.213,E2 -12807.213} C_VEL
LIN {X 0,Y 368.879,Z 385.153,A -85,B 0,C 180,E1 -12809.694,E2 -12809.694} C_VEL
LIN {X 0,Y 368.882,Z 385.159,A -85,B 0,C 180,E1 -12813.54,E2 -12813.54} C_VEL
LIN {X 0,Y 368.883,Z 385.129,A -85,B 0,C 180,E1 -12816.856,E2 -12816.856} C_VEL
LIN {X 0,Y 368.872,Z 385.164,A -85,B 0,C 180,E1 -12820.375,E2 -12820.375} C_VEL
LIN {X 0,Y 368.867,Z 385.144,A -85,B 0,C 180,E1 -12823.617,E2 -12823.617} C_VEL
LIN {X 0,Y 368.899,Z 385.293,A -85,B 0,C 180,E1 -12826.493,E2 -12826.493} C_VEL
LIN {X 0,Y 369.11,Z 386.219,A -85,B 0,C 180,E1 -12826.732,E2 -12826.732} C_VEL
LIN {X 0,Y 373.973,Z 398.839,A -85,B 0,C 180,E1 -12829.149,E2 -12829.149} C_VEL
LIN {X 0,Y 378.944,Z 413.962,A -85,B 0,C 180,E1 -12831.85,E2 -12831.85} C_VEL
LIN {X 0,Y 383.175,Z 428.874,A -85,B 0,C 180,E1 -12834.35,E2 -12834.35} C_VEL
LIN {X 0,Y 383.999,Z 432.836,A -85,B 0,C 180,E1 -12834.97,E2 -12834.97} C_VEL
LIN {X 0,Y 381.799,Z 459.563,A -85,B 0,C 180,E1 -12838.28,E2 -12838.28} C_VEL
LIN {X 0,Y 381.048,Z 471.604,A -85,B 0,C 180,E1 -12839.679,E2 -12839.679} C_VEL
LIN {X 0,Y 386.399,Z 505.055,A -85,B 0,C 180,E1 -12840.852,E2 -12840.852} C_VEL
LIN {X 0,Y 384.629,Z 585.302,A -85,B 0,C 180,E1 -12842.379,E2 -12842.379} C_VEL
LIN {X 0,Y 383.198,Z 640.752,A -85,B 0,C 180,E1 -12843.448,E2 -12843.448} C_VEL
LIN {X 0,Y 382.414,Z 656.07,A -85,B 0,C 180,E1 -12843.935,E2 -12843.935} C_VEL
LIN {X 0,Y 381.364,Z 669.754,A -85,B 0,C 180,E1 -12844.555,E2 -12844.555} C_VEL
LIN {X 0,Y 380.023,Z 684.031,A -85,B 0,C 180,E1 -12845.413,E2 -12845.413} C_VEL
LIN {X 0,Y 378.469,Z 697.854,A -85,B 0,C 180,E1 -12846.471,E2 -12846.471} C_VEL
LIN {X 0,Y 376.864,Z 710.536,A -85,B 0,C 180,E1 -12847.671,E2 -12847.671} C_VEL
LIN {X 0,Y 375.252,Z 722.278,A -85,B 0,C 180,E1 -12849.013,E2 -12849.013} C_VEL
LIN {X 0,Y 373.712,Z 733.166,A -85,B 0,C 180,E1 -12850.502,E2 -12850.502} C_VEL
LIN {X 0,Y 372.179,Z 743.203,A -85,B 0,C 180,E1 -12852.132,E2 -12852.132} C_VEL
LIN {X 0,Y 370.749,Z 753.01,A -85,B 0,C 180,E1 -12854.048,E2 -12854.048} C_VEL
LIN {X 0,Y 369.69,Z 760.551,A -85,B 0,C 180,E1 -12855.822,E2 -12855.822} C_VEL
LIN {X 0,Y 368.823,Z 767.895,A -85,B 0,C 180,E1 -12857.903,E2 -12857.903} C_VEL
LIN {X 0,Y 368.085,Z 774.148,A -85,B 0,C 180,E1 -12860.107,E2 -12860.107} C_VEL
LIN {X 0,Y 367.658,Z 778.981,A -85,B 0,C 180,E1 -12862.312,E2 -12862.312} C_VEL
LIN {X 0,Y 367.434,Z 782.523,A -85,B 0,C 180,E1 -12864.514,E2 -12864.514} C_VEL
LIN {X 0,Y 367.34,Z 784.865,A -85,B 0,C 180,E1 -12866.711,E2 -12866.711} C_VEL
LIN {X 0,Y 367.347,Z 786.058,A -85,B 0,C 180,E1 -12868.905,E2 -12868.905} C_VEL
LIN {X 0,Y 367.348,Z 786.072,A -85,B 0,C 180,E1 -12871.098,E2 -12871.098} C_VEL
LIN {X 0,Y 367.341,Z 784.938,A -85,B 0,C 180,E1 -12873.292,E2 -12873.292} C_VEL
LIN {X 0,Y 367.41,Z 783.37,A -85,B 0,C 180,E1 -12874.877,E2 -12874.877} C_VEL
LIN {X 0,Y 366.784,Z 782.299,A -85,B 0,C 180,E1 -12875.778,E2 -12875.778} C_VEL
LIN {X 0,Y 364.041,Z 780.144,A -85,B 0,C 180,E1 -12877.237,E2 -12877.237} C_VEL
LIN {X 0,Y 361.785,Z 778.091,A -85,B 0,C 180,E1 -12878.402,E2 -12878.402} C_VEL
LIN {X 0,Y 360.92,Z 776.25,A -85,B 0,C 180,E1 -12879.287,E2 -12879.287} C_VEL
LIN {X 0,Y 360.905,Z 775.572,A -85,B 0,C 180,E1 -12879.583,E2 -12879.583} C_VEL
LIN {X 0,Y 361.57,Z 769.872,A -85,B 0,C 180,E1 -12881.778,E2 -12881.778} C_VEL
LIN {X 0,Y 362.558,Z 762.373,A -85,B 0,C 180,E1 -12884.067,E2 -12884.067} C_VEL
LIN {X 0,Y 363.81,Z 753.417,A -85,B 0,C 180,E1 -12886.268,E2 -12886.268} C_VEL
LIN {X 0,Y 365.296,Z 743.695,A -85,B 0,C 180,E1 -12888.22,E2 -12888.22} C_VEL
LIN {X 0,Y 366.865,Z 733.734,A -85,B 0,C 180,E1 -12889.881,E2 -12889.881} C_VEL
LIN {X 0,Y 368.626,Z 721.902,A -85,B 0,C 180,E1 -12891.533,E2 -12891.533} C_VEL
LIN {X 0,Y 370.513,Z 708.822,A -85,B 0,C 180,E1 -12893.032,E2 -12893.032} C_VEL
LIN {X 0,Y 372.221,Z 695.776,A -85,B 0,C 180,E1 -12894.248,E2 -12894.248} C_VEL
LIN {X 0,Y 373.832,Z 681.872,A -85,B 0,C 180,E1 -12895.289,E2 -12895.289} C_VEL
LIN {X 0,Y 375.182,Z 667.297,A -85,B 0,C 180,E1 -12896.141,E2 -12896.141} C_VEL
LIN {X 0,Y 376.369,Z 651.484,A -85,B 0,C 180,E1 -12896.814,E2 -12896.814} C_VEL
LIN {X 0,Y 377.094,Z 636.062,A -85,B 0,C 180,E1 -12897.245,E2 -12897.245} C_VEL
LIN {X 0,Y 379.836,Z 526.323,A -85,B 0,C 180,E1 -12899.349,E2 -12899.349} C_VEL
LIN {X 0,Y 380.262,Z 506.161,A -85,B 0,C 180,E1 -12899.743,E2 -12899.743} C_VEL
LIN {X 0,Y 374.701,Z 471.242,A -85,B 0,C 180,E1 -12901.013,E2 -12901.013} C_VEL
LIN {X 0,Y 376.11,Z 452.357,A -85,B 0,C 180,E1 -12903.293,E2 -12903.293} C_VEL
LIN {X 0,Y 377.623,Z 435.068,A -85,B 0,C 180,E1 -12905.479,E2 -12905.479} C_VEL
LIN {X 0,Y 374.811,Z 424.103,A -85,B 0,C 180,E1 -12907.285,E2 -12907.285} C_VEL
LIN {X 0,Y 370.467,Z 409.756,A -85,B 0,C 180,E1 -12909.798,E2 -12909.798} C_VEL
LIN {X 0,Y 365.815,Z 396.678,A -85,B 0,C 180,E1 -12912.255,E2 -12912.255} C_VEL
LIN {X 0,Y 361.84,Z 386.292,A -85,B 0,C 180,E1 -12914.367,E2 -12914.367} C_VEL
LIN {X 0,Y 361.798,Z 386.022,A -85,B 0,C 180,E1 -12915.952,E2 -12915.952} C_VEL
LIN {X 0,Y 361.814,Z 386.017,A -85,B 0,C 180,E1 -12919.25,E2 -12919.25} C_VEL
LIN {X 0,Y 361.865,Z 386.032,A -85,B 0,C 180,E1 -12922.982,E2 -12922.982} C_VEL
LIN {X 0,Y 361.862,Z 386.015,A -85,B 0,C 180,E1 -12926.632,E2 -12926.632} C_VEL
LIN {X 0,Y 361.852,Z 386.038,A -85,B 0,C 180,E1 -12929.67,E2 -12929.67} C_VEL
LIN {X 0,Y 361.842,Z 386.167,A -85,B 0,C 180,E1 -12933.081,E2 -12933.081} C_VEL
LIN {X 0,Y 363.009,Z 390.746,A -85,B 0,C 180,E1 -12934.097,E2 -12934.097} C_VEL
LIN {X 0,Y 373.007,Z 417.086,A -85,B 0,C 180,E1 -12935.419,E2 -12935.419} C_VEL
LIN {X 0,Y 369.439,Z 533.478,A -85,B 0,C 180,E1 -12938.372,E2 -12938.372} C_VEL
LIN {X 0,Y 369.004,Z 549.153,A -85,B 0,C 180,E1 -12938.997,E2 -12938.997} C_VEL
LIN {X 0,Y 368.411,Z 563.753,A -85,B 0,C 180,E1 -12939.801,E2 -12939.801} C_VEL
LIN {X 0,Y 367.63,Z 577.111,A -85,B 0,C 180,E1 -12940.745,E2 -12940.745} C_VEL
LIN {X 0,Y 366.889,Z 589.809,A -85,B 0,C 180,E1 -12941.864,E2 -12941.864} C_VEL
LIN {X 0,Y 365.964,Z 602.734,A -85,B 0,C 180,E1 -12943.258,E2 -12943.258} C_VEL
LIN {X 0,Y 365.227,Z 613.455,A -85,B 0,C 180,E1 -12944.657,E2 -12944.657} C_VEL
LIN {X 0,Y 364.329,Z 624.156,A -85,B 0,C 180,E1 -12946.331,E2 -12946.331} C_VEL
LIN {X 0,Y 363.702,Z 633.057,A -85,B 0,C 180,E1 -12948.011,E2 -12948.011} C_VEL
LIN {X 0,Y 363.103,Z 641.621,A -85,B 0,C 180,E1 -12949.968,E2 -12949.968} C_VEL
LIN {X 0,Y 362.713,Z 648.277,A -85,B 0,C 180,E1 -12951.844,E2 -12951.844} C_VEL
LIN {X 0,Y 362.357,Z 654.039,A -85,B 0,C 180,E1 -12953.876,E2 -12953.876} C_VEL
LIN {X 0,Y 361.955,Z 657.726,A -85,B 0,C 180,E1 -12955.545,E2 -12955.545} C_VEL
LIN {X 0,Y 362.131,Z 659.682,A -85,B 0,C 180,E1 -12956.662,E2 -12956.662} C_VEL
LIN {X 0,Y 362.077,Z 662.544,A -85,B 0,C 180,E1 -12958.888,E2 -12958.888} C_VEL
LIN {X 0,Y 362.275,Z 663.951,A -85,B 0,C 180,E1 -12961.111,E2 -12961.111} C_VEL
LIN {X 0,Y 362.729,Z 663.887,A -85,B 0,C 180,E1 -12963.332,E2 -12963.332} C_VEL
LIN {X 0,Y 363.182,Z 662.437,A -85,B 0,C 180,E1 -12965.552,E2 -12965.552} C_VEL
LIN {X 0,Y 363.996,Z 659.503,A -85,B 0,C 180,E1 -12967.767,E2 -12967.767} C_VEL
LIN {X 0,Y 364.817,Z 656.291,A -85,B 0,C 180,E1 -12969.424,E2 -12969.424} C_VEL
LIN {X 0,Y 365.978,Z 650.503,A -85,B 0,C 180,E1 -12971.653,E2 -12971.653} C_VEL
LIN {X 0,Y 367.294,Z 644.039,A -85,B 0,C 180,E1 -12973.556,E2 -12973.556} C_VEL
LIN {X 0,Y 368.792,Z 635.87,A -85,B 0,C 180,E1 -12975.474,E2 -12975.474} C_VEL
LIN {X 0,Y 370.526,Z 625.726,A -85,B 0,C 180,E1 -12977.382,E2 -12977.382} C_VEL
LIN {X 0,Y 372.218,Z 615.156,A -85,B 0,C 180,E1 -12978.987,E2 -12978.987} C_VEL
LIN {X 0,Y 373.854,Z 603.068,A -85,B 0,C 180,E1 -12980.495,E2 -12980.495} C_VEL
LIN {X 0,Y 375.291,Z 591.29,A -85,B 0,C 180,E1 -12981.707,E2 -12981.707} C_VEL
LIN {X 0,Y 376.683,Z 578.337,A -85,B 0,C 180,E1 -12982.777,E2 -12982.777} C_VEL
LIN {X 0,Y 377.86,Z 564.088,A -85,B 0,C 180,E1 -12983.715,E2 -12983.715} C_VEL
LIN {X 0,Y 378.897,Z 548.772,A -85,B 0,C 180,E1 -12984.487,E2 -12984.487} C_VEL
LIN {X 0,Y 379.896,Z 529.702,A -85,B 0,C 180,E1 -12985.182,E2 -12985.182} C_VEL
LIN {X 0,Y 385.98,Z 461.431,A -85,B 0,C 180,E1 -12987.466,E2 -12987.466} C_VEL
LIN {X 0,Y 388.481,Z 436.451,A -85,B 0,C 180,E1 -12988.321,E2 -12988.321} C_VEL
LIN {X 0,Y 384.36,Z 429.427,A -85,B 0,C 180,E1 -12989.446,E2 -12989.446} C_VEL
LIN {X 0,Y 380.697,Z 423.962,A -85,B 0,C 180,E1 -12990.508,E2 -12990.508} C_VEL
LIN {X 0,Y 377.78,Z 420.087,A -85,B 0,C 180,E1 -12991.422,E2 -12991.422} C_VEL
LIN {X 0,Y 375.157,Z 416.768,A -85,B 0,C 180,E1 -12992.321,E2 -12992.321} C_VEL
LIN {X 0,Y 373.14,Z 414.026,A -85,B 0,C 180,E1 -12993.173,E2 -12993.173} C_VEL
LIN {X 0,Y 372.378,Z 411.258,A -85,B 0,C 180,E1 -12995.808,E2 -12995.808} C_VEL
LIN {X 0,Y 372.066,Z 409.909,A -85,B 0,C 180,E1 -12998.56,E2 -12998.56} C_VEL
LIN {X 0,Y 372.222,Z 410.004,A -85,B 0,C 180,E1 -13000.951,E2 -13000.951} C_VEL
LIN {X 0,Y 372.665,Z 410.841,A -85,B 0,C 180,E1 -13002.759,E2 -13002.759} C_VEL
LIN {X 0,Y 373.353,Z 412.166,A -85,B 0,C 180,E1 -13004.33,E2 -13004.33} C_VEL
LIN {X 0,Y 374.199,Z 414.278,A -85,B 0,C 180,E1 -13005.978,E2 -13005.978} C_VEL
LIN {X 0,Y 375.838,Z 418.622,A -85,B 0,C 180,E1 -13008.416,E2 -13008.416} C_VEL
LIN {X 0,Y 377.606,Z 424.337,A -85,B 0,C 180,E1 -13010.741,E2 -13010.741} C_VEL
LIN {X 0,Y 379.279,Z 430.926,A -85,B 0,C 180,E1 -13012.824,E2 -13012.824} C_VEL
LIN {X 0,Y 380.451,Z 436.737,A -85,B 0,C 180,E1 -13014.371,E2 -13014.371} C_VEL
LIN {X 0,Y 380.558,Z 438.077,A -85,B 0,C 180,E1 -13014.684,E2 -13014.684} C_VEL
LIN {X 0,Y 379.183,Z 444.324,A -85,B 0,C 180,E1 -13015.696,E2 -13015.696} C_VEL
LIN {X 0,Y 381.387,Z 461.001,A -85,B 0,C 180,E1 -13016.984,E2 -13016.984} C_VEL
LIN {X 0,Y 383.192,Z 478.779,A -85,B 0,C 180,E1 -13018.116,E2 -13018.116} C_VEL
LIN {X 0,Y 384.04,Z 492.626,A -85,B 0,C 180,E1 -13018.85,E2 -13018.85} C_VEL
LIN {X 0,Y 384.384,Z 505.848,A -85,B 0,C 180,E1 -13019.449,E2 -13019.449} C_VEL
LIN {X 0,Y 379.62,Z 574.204,A -85,B 0,C 180,E1 -13021.452,E2 -13021.452} C_VEL
LIN {X 0,Y 377.051,Z 616.799,A -85,B 0,C 180,E1 -13022.639,E2 -13022.639} C_VEL
LIN {X 0,Y 376.228,Z 643.009,A -85,B 0,C 180,E1 -13023.175,E2 -13023.175} C_VEL
LIN {X 0,Y 375.321,Z 658.371,A -85,B 0,C 180,E1 -13023.705,E2 -13023.705} C_VEL
LIN {X 0,Y 374.173,Z 672.623,A -85,B 0,C 180,E1 -13024.404,E2 -13024.404} C_VEL
LIN {X 0,Y 372.784,Z 687.292,A -85,B 0,C 180,E1 -13025.365,E2 -13025.365} C_VEL
LIN {X 0,Y 371.201,Z 700.216,A -85,B 0,C 180,E1 -13026.423,E2 -13026.423} C_VEL
LIN {X 0,Y 369.424,Z 713.573,A -85,B 0,C 180,E1 -13027.782,E2 -13027.782} C_VEL
LIN {X 0,Y 367.641,Z 725.716,A -85,B 0,C 180,E1 -13029.288,E2 -13029.288} C_VEL
LIN {X 0,Y 366.065,Z 736.776,A -85,B 0,C 180,E1 -13030.949,E2 -13030.949} C_VEL
LIN {X 0,Y 364.598,Z 746.078,A -85,B 0,C 180,E1 -13032.614,E2 -13032.614} C_VEL
LIN {X 0,Y 363.259,Z 755.204,A -85,B 0,C 180,E1 -13034.571,E2 -13034.571} C_VEL
LIN {X 0,Y 362.185,Z 762.77,A -85,B 0,C 180,E1 -13036.533,E2 -13036.533} C_VEL
LIN {X 0,Y 361.571,Z 768.214,A -85,B 0,C 180,E1 -13038.222,E2 -13038.222} C_VEL
LIN {X 0,Y 360.924,Z 774.117,A -85,B 0,C 180,E1 -13040.471,E2 -13040.471} C_VEL
LIN {X 0,Y 360.655,Z 777.605,A -85,B 0,C 180,E1 -13042.158,E2 -13042.158} C_VEL
LIN {X 0,Y 360.45,Z 781.149,A -85,B 0,C 180,E1 -13044.404,E2 -13044.404} C_VEL
LIN {X 0,Y 360.345,Z 783.477,A -85,B 0,C 180,E1 -13046.644,E2 -13046.644} C_VEL
LIN {X 0,Y 360.331,Z 784.645,A -85,B 0,C 180,E1 -13048.881,E2 -13048.881} C_VEL
LIN {X 0,Y 360.333,Z 784.643,A -85,B 0,C 180,E1 -13051.116,E2 -13051.116} C_VEL
LIN {X 0,Y 360.348,Z 783.469,A -85,B 0,C 180,E1 -13053.353,E2 -13053.353} C_VEL
LIN {X 0,Y 360.434,Z 781.137,A -85,B 0,C 180,E1 -13055.593,E2 -13055.593} C_VEL
LIN {X 0,Y 360.651,Z 777.595,A -85,B 0,C 180,E1 -13057.838,E2 -13057.838} C_VEL
LIN {X 0,Y 361.048,Z 772.75,A -85,B 0,C 180,E1 -13060.088,E2 -13060.088} C_VEL
LIN {X 0,Y 361.787,Z 766.471,A -85,B 0,C 180,E1 -13062.336,E2 -13062.336} C_VEL
LIN {X 0,Y 362.735,Z 758.577,A -85,B 0,C 180,E1 -13064.587,E2 -13064.587} C_VEL
LIN {X 0,Y 363.952,Z 750.147,A -85,B 0,C 180,E1 -13066.546,E2 -13066.546} C_VEL
LIN {X 0,Y 365.447,Z 739.972,A -85,B 0,C 180,E1 -13068.499,E2 -13068.499} C_VEL
LIN {X 0,Y 367.034,Z 729.544,A -85,B 0,C 180,E1 -13070.159,E2 -13070.159} C_VEL
LIN {X 0,Y 368.68,Z 718.182,A -85,B 0,C 180,E1 -13071.673,E2 -13071.673} C_VEL
LIN {X 0,Y 370.399,Z 705.802,A -85,B 0,C 180,E1 -13073.036,E2 -13073.036} C_VEL
LIN {X 0,Y 372.129,Z 692.209,A -85,B 0,C 180,E1 -13074.251,E2 -13074.251} C_VEL
LIN {X 0,Y 373.56,Z 679.02,A -85,B 0,C 180,E1 -13075.201,E2 -13075.201} C_VEL
LIN {X 0,Y 374.843,Z 664.496,A -85,B 0,C 180,E1 -13076.013,E2 -13076.013} C_VEL
LIN {X 0,Y 375.843,Z 649.515,A -85,B 0,C 180,E1 -13076.622,E2 -13076.622} C_VEL
LIN {X 0,Y 376.5,Z 634.238,A -85,B 0,C 180,E1 -13077.025,E2 -13077.025} C_VEL
LIN {X 0,Y 379.328,Z 517.024,A -85,B 0,C 180,E1 -13079.265,E2 -13079.265} C_VEL
LIN {X 0,Y 379.481,Z 502.729,A -85,B 0,C 180,E1 -13079.555,E2 -13079.555} C_VEL
LIN {X 0,Y 375.299,Z 469.867,A -85,B 0,C 180,E1 -13080.631,E2 -13080.631} C_VEL
LIN {X 0,Y 374.601,Z 464.29,A -85,B 0,C 180,E1 -13080.878,E2 -13080.878} C_VEL
LIN {X 0,Y 372.797,Z 435.903,A -85,B 0,C 180,E1 -13082.616,E2 -13082.616} C_VEL
LIN {X 0,Y 373.688,Z 427.586,A -85,B 0,C 180,E1 -13083.741,E2 -13083.741} C_VEL
LIN {X 0,Y 368.593,Z 409.11,A -85,B 0,C 180,E1 -13086.792,E2 -13086.792} C_VEL
LIN {X 0,Y 362.95,Z 389.967,A -85,B 0,C 180,E1 -13090.162,E2 -13090.162} C_VEL
LIN {X 0,Y 361.855,Z 386.169,A -85,B 0,C 180,E1 -13090.925,E2 -13090.925} C_VEL
LIN {X 0,Y 361.803,Z 386.044,A -85,B 0,C 180,E1 -13094.368,E2 -13094.368} C_VEL
LIN {X 0,Y 361.81,Z 386,A -85,B 0,C 180,E1 -13097.569,E2 -13097.569} C_VEL
LIN {X 0,Y 361.829,Z 386.039,A -85,B 0,C 180,E1 -13101.571,E2 -13101.571} C_VEL
LIN {X 0,Y 361.856,Z 385.985,A -85,B 0,C 180,E1 -13104.655,E2 -13104.655} C_VEL
LIN {X 0,Y 361.824,Z 386.04,A -85,B 0,C 180,E1 -13108.369,E2 -13108.369} C_VEL
LIN {X 0,Y 361.852,Z 386.023,A -85,B 0,C 180,E1 -13110.951,E2 -13110.951} C_VEL
LIN {X 0,Y 361.847,Z 386.022,A -85,B 0,C 180,E1 -13114.704,E2 -13114.704} C_VEL
LIN {X 0,Y 361.839,Z 386.035,A -85,B 0,C 180,E1 -13118.344,E2 -13118.344} C_VEL
LIN {X 0,Y 361.889,Z 386.03,A -85,B 0,C 180,E1 -13122.092,E2 -13122.092} C_VEL
LIN {X 0,Y 361.964,Z 386.009,A -85,B 0,C 180,E1 -13126.113,E2 -13126.113} C_VEL
LIN {X 0,Y 361.981,Z 386.004,A -85,B 0,C 180,E1 -13129.937,E2 -13129.937} C_VEL
LIN {X 0,Y 362.1,Z 386.003,A -85,B 0,C 180,E1 -13133.313,E2 -13133.313} C_VEL
LIN {X 0,Y 362.252,Z 385.982,A -85,B 0,C 180,E1 -13137.776,E2 -13137.776} C_VEL
LIN {X 0,Y 362.249,Z 385.973,A -85,B 0,C 180,E1 -13142.224,E2 -13142.224} C_VEL
LIN {X 0,Y 362.125,Z 385.985,A -85,B 0,C 180,E1 -13146.687,E2 -13146.687} C_VEL
LIN {X 0,Y 361.982,Z 386.017,A -85,B 0,C 180,E1 -13150.064,E2 -13150.064} C_VEL
LIN {X 0,Y 361.983,Z 386.016,A -85,B 0,C 180,E1 -13153.899,E2 -13153.899} C_VEL
LIN {X 0,Y 361.913,Z 386.013,A -85,B 0,C 180,E1 -13156.935,E2 -13156.935} C_VEL
LIN {X 0,Y 361.869,Z 386.023,A -85,B 0,C 180,E1 -13160.462,E2 -13160.462} C_VEL
LIN {X 0,Y 361.847,Z 386.036,A -85,B 0,C 180,E1 -13164.102,E2 -13164.102} C_VEL
LIN {X 0,Y 361.821,Z 386.04,A -85,B 0,C 180,E1 -13167.786,E2 -13167.786} C_VEL
LIN {X 0,Y 361.813,Z 386.043,A -85,B 0,C 180,E1 -13171.281,E2 -13171.281} C_VEL
LIN {X 0,Y 361.838,Z 386.041,A -85,B 0,C 180,E1 -13174.282,E2 -13174.282} C_VEL
LIN {X 0,Y 361.845,Z 386.003,A -85,B 0,C 180,E1 -13177.223,E2 -13177.223} C_VEL
LIN {X 0,Y 361.798,Z 386.038,A -85,B 0,C 180,E1 -13180.752,E2 -13180.752} C_VEL
LIN {X 0,Y 361.8,Z 386.038,A -85,B 0,C 180,E1 -13184.371,E2 -13184.371} C_VEL
LIN {X 0,Y 361.849,Z 386.248,A -85,B 0,C 180,E1 -13185.74,E2 -13185.74} C_VEL
LIN {X 0,Y 366.2,Z 397.612,A -85,B 0,C 180,E1 -13188.029,E2 -13188.029} C_VEL
LIN {X 0,Y 370.869,Z 411.106,A -85,B 0,C 180,E1 -13190.553,E2 -13190.553} C_VEL
LIN {X 0,Y 375.43,Z 426.287,A -85,B 0,C 180,E1 -13193.202,E2 -13193.202} C_VEL
LIN {X 0,Y 377.576,Z 434.574,A -85,B 0,C 180,E1 -13194.569,E2 -13194.569} C_VEL
LIN {X 0,Y 375.611,Z 458.452,A -85,B 0,C 180,E1 -13197.571,E2 -13197.571} C_VEL
LIN {X 0,Y 374.704,Z 471.222,A -85,B 0,C 180,E1 -13199.092,E2 -13199.092} C_VEL
LIN {X 0,Y 379.899,Z 504.25,A -85,B 0,C 180,E1 -13200.289,E2 -13200.289} C_VEL
LIN {X 0,Y 380.28,Z 508.17,A -85,B 0,C 180,E1 -13200.405,E2 -13200.405} C_VEL
LIN {X 0,Y 376.939,Z 639.304,A -85,B 0,C 180,E1 -13202.934,E2 -13202.934} C_VEL
LIN {X 0,Y 376.134,Z 654.487,A -85,B 0,C 180,E1 -13203.4,E2 -13203.4} C_VEL
LIN {X 0,Y 374.975,Z 669.499,A -85,B 0,C 180,E1 -13204.077,E2 -13204.077} C_VEL
LIN {X 0,Y 373.566,Z 684.001,A -85,B 0,C 180,E1 -13204.959,E2 -13204.959} C_VEL
LIN {X 0,Y 371.956,Z 697.828,A -85,B 0,C 180,E1 -13206.034,E2 -13206.034} C_VEL
LIN {X 0,Y 370.275,Z 710.514,A -85,B 0,C 180,E1 -13207.251,E2 -13207.251} C_VEL
LIN {X 0,Y 368.579,Z 722.258,A -85,B 0,C 180,E1 -13208.615,E2 -13208.615} C_VEL
LIN {X 0,Y 366.991,Z 733.148,A -85,B 0,C 180,E1 -13210.13,E2 -13210.13} C_VEL
LIN {X 0,Y 365.382,Z 743.186,A -85,B 0,C 180,E1 -13211.788,E2 -13211.788} C_VEL
LIN {X 0,Y 363.877,Z 752.995,A -85,B 0,C 180,E1 -13213.738,E2 -13213.738} C_VEL
LIN {X 0,Y 362.589,Z 761.945,A -85,B 0,C 180,E1 -13215.913,E2 -13215.913} C_VEL
LIN {X 0,Y 361.593,Z 769.599,A -85,B 0,C 180,E1 -13218.226,E2 -13218.226} C_VEL
LIN {X 0,Y 360.906,Z 775.492,A -85,B 0,C 180,E1 -13220.474,E2 -13220.474} C_VEL
LIN {X 0,Y 360.592,Z 778.968,A -85,B 0,C 180,E1 -13222.16,E2 -13222.16} C_VEL
LIN {X 0,Y 360.337,Z 782.51,A -85,B 0,C 180,E1 -13224.405,E2 -13224.405} C_VEL
LIN {X 0,Y 360.261,Z 784.852,A -85,B 0,C 180,E1 -13226.647,E2 -13226.647} C_VEL
LIN {X 0,Y 360.245,Z 786.044,A -85,B 0,C 180,E1 -13228.884,E2 -13228.884} C_VEL
LIN {X 0,Y 360.246,Z 786.058,A -85,B 0,C 180,E1 -13231.12,E2 -13231.12} C_VEL
LIN {X 0,Y 360.262,Z 784.923,A -85,B 0,C 180,E1 -13233.357,E2 -13233.357} C_VEL
LIN {X 0,Y 360.357,Z 782.637,A -85,B 0,C 180,E1 -13235.598,E2 -13235.598} C_VEL
LIN {X 0,Y 360.629,Z 779.146,A -85,B 0,C 180,E1 -13237.842,E2 -13237.842} C_VEL
LIN {X 0,Y 360.905,Z 775.572,A -85,B 0,C 180,E1 -13239.583,E2 -13239.583} C_VEL
LIN {X 0,Y 360.466,Z 773.512,A -85,B 0,C 180,E1 -13240.458,E2 -13240.458} C_VEL
LIN {X 0,Y 358.057,Z 769.9,A -85,B 0,C 180,E1 -13241.882,E2 -13241.882} C_VEL
LIN {X 0,Y 355.761,Z 765.889,A -85,B 0,C 180,E1 -13243.294,E2 -13243.294} C_VEL
LIN {X 0,Y 355.51,Z 763.086,A -85,B 0,C 180,E1 -13244.138,E2 -13244.138} C_VEL
LIN {X 0,Y 356.744,Z 754.612,A -85,B 0,C 180,E1 -13246.305,E2 -13246.305} C_VEL
LIN {X 0,Y 358.226,Z 745.138,A -85,B 0,C 180,E1 -13248.296,E2 -13248.296} C_VEL
LIN {X 0,Y 359.853,Z 735.569,A -85,B 0,C 180,E1 -13249.969,E2 -13249.969} C_VEL
LIN {X 0,Y 361.633,Z 723.975,A -85,B 0,C 180,E1 -13251.671,E2 -13251.671} C_VEL
LIN {X 0,Y 363.637,Z 711.319,A -85,B 0,C 180,E1 -13253.192,E2 -13253.192} C_VEL
LIN {X 0,Y 365.33,Z 698.823,A -85,B 0,C 180,E1 -13254.433,E2 -13254.433} C_VEL
LIN {X 0,Y 366.987,Z 685.979,A -85,B 0,C 180,E1 -13255.467,E2 -13255.467} C_VEL
LIN {X 0,Y 368.361,Z 672.32,A -85,B 0,C 180,E1 -13256.352,E2 -13256.352} C_VEL
LIN {X 0,Y 369.613,Z 657.629,A -85,B 0,C 180,E1 -13257.069,E2 -13257.069} C_VEL
LIN {X 0,Y 370.523,Z 642.79,A -85,B 0,C 180,E1 -13257.578,E2 -13257.578} C_VEL
LIN {X 0,Y 371.633,Z 607.58,A -85,B 0,C 180,E1 -13258.293,E2 -13258.293} C_VEL
LIN {X 0,Y 374.109,Z 507.49,A -85,B 0,C 180,E1 -13260.25,E2 -13260.25} C_VEL
LIN {X 0,Y 368.565,Z 472.512,A -85,B 0,C 180,E1 -13261.532,E2 -13261.532} C_VEL
LIN {X 0,Y 368.42,Z 470.201,A -85,B 0,C 180,E1 -13261.707,E2 -13261.707} C_VEL
LIN {X 0,Y 370.198,Z 448.495,A -85,B 0,C 180,E1 -13264.389,E2 -13264.389} C_VEL
LIN {X 0,Y 371.167,Z 438.316,A -85,B 0,C 180,E1 -13265.692,E2 -13265.692} C_VEL
LIN {X 0,Y 370.714,Z 435.03,A -85,B 0,C 180,E1 -13266.196,E2 -13266.196} C_VEL
LIN {X 0,Y 366.189,Z 418.803,A -85,B 0,C 180,E1 -13268.988,E2 -13268.988} C_VEL
LIN {X 0,Y 361.661,Z 405.147,A -85,B 0,C 180,E1 -13271.526,E2 -13271.526} C_VEL
LIN {X 0,Y 357.464,Z 394.051,A -85,B 0,C 180,E1 -13273.75,E2 -13273.75} C_VEL
LIN {X 0,Y 354.819,Z 387.137,A -85,B 0,C 180,E1 -13275.209,E2 -13275.209} C_VEL
LIN {X 0,Y 354.771,Z 386.899,A -85,B 0,C 180,E1 -13278.833,E2 -13278.833} C_VEL
LIN {X 0,Y 354.803,Z 386.916,A -85,B 0,C 180,E1 -13282.405,E2 -13282.405} C_VEL
LIN {X 0,Y 354.812,Z 386.88,A -85,B 0,C 180,E1 -13284.941,E2 -13284.941} C_VEL
LIN {X 0,Y 354.781,Z 386.918,A -85,B 0,C 180,E1 -13288.41,E2 -13288.41} C_VEL
LIN {X 0,Y 354.794,Z 386.918,A -85,B 0,C 180,E1 -13291.614,E2 -13291.614} C_VEL
LIN {X 0,Y 354.807,Z 387.095,A -85,B 0,C 180,E1 -13292.738,E2 -13292.738} C_VEL
LIN {X 0,Y 355.819,Z 391.217,A -85,B 0,C 180,E1 -13293.667,E2 -13293.667} C_VEL
LIN {X 0,Y 366.192,Z 418.504,A -85,B 0,C 180,E1 -13295.077,E2 -13295.077} C_VEL
LIN {X 0,Y 363.029,Z 514.497,A -85,B 0,C 180,E1 -13297.558,E2 -13297.558} C_VEL
LIN {X 0,Y 362.474,Z 537.046,A -85,B 0,C 180,E1 -13298.197,E2 -13298.197} C_VEL
LIN {X 0,Y 362.058,Z 552.72,A -85,B 0,C 180,E1 -13298.878,E2 -13298.878} C_VEL
LIN {X 0,Y 361.385,Z 567.185,A -85,B 0,C 180,E1 -13299.732,E2 -13299.732} C_VEL
LIN {X 0,Y 360.539,Z 581.134,A -85,B 0,C 180,E1 -13300.795,E2 -13300.795} C_VEL
LIN {X 0,Y 359.696,Z 594.591,A -85,B 0,C 180,E1 -13302.077,E2 -13302.077} C_VEL
LIN {X 0,Y 358.723,Z 607.303,A -85,B 0,C 180,E1 -13303.555,E2 -13303.555} C_VEL
LIN {X 0,Y 358.04,Z 617.075,A -85,B 0,C 180,E1 -13304.925,E2 -13304.925} C_VEL
LIN {X 0,Y 357.126,Z 627.386,A -85,B 0,C 180,E1 -13306.63,E2 -13306.63} C_VEL
LIN {X 0,Y 356.553,Z 635.958,A -85,B 0,C 180,E1 -13308.344,E2 -13308.344} C_VEL
LIN {X 0,Y 355.967,Z 644.182,A -85,B 0,C 180,E1 -13310.339,E2 -13310.339} C_VEL
LIN {X 0,Y 355.617,Z 649.98,A -85,B 0,C 180,E1 -13312.048,E2 -13312.048} C_VEL
LIN {X 0,Y 355.346,Z 654.695,A -85,B 0,C 180,E1 -13313.755,E2 -13313.755} C_VEL
LIN {X 0,Y 355.002,Z 659.61,A -85,B 0,C 180,E1 -13316.027,E2 -13316.027} C_VEL
LIN {X 0,Y 354.989,Z 662.215,A -85,B 0,C 180,E1 -13317.731,E2 -13317.731} C_VEL
LIN {X 0,Y 355.072,Z 664.462,A -85,B 0,C 180,E1 -13320,E2 -13320} C_VEL
LIN {X 0,Y 355.481,Z 665.276,A -85,B 0,C 180,E1 -13322.266,E2 -13322.266} C_VEL
LIN {X 0,Y 356.001,Z 664.644,A -85,B 0,C 180,E1 -13324.529,E2 -13324.529} C_VEL
LIN {X 0,Y 356.6,Z 662.58,A -85,B 0,C 180,E1 -13326.791,E2 -13326.791} C_VEL
LIN {X 0,Y 357.639,Z 659.014,A -85,B 0,C 180,E1 -13329.045,E2 -13329.045} C_VEL
LIN {X 0,Y 358.6,Z 655.32,A -85,B 0,C 180,E1 -13330.73,E2 -13330.73} C_VEL
LIN {X 0,Y 359.645,Z 650.65,A -85,B 0,C 180,E1 -13332.413,E2 -13332.413} C_VEL
LIN {X 0,Y 361.097,Z 643.824,A -85,B 0,C 180,E1 -13334.368,E2 -13334.368} C_VEL
LIN {X 0,Y 362.538,Z 636.686,A -85,B 0,C 180,E1 -13336.036,E2 -13336.036} C_VEL
LIN {X 0,Y 364.102,Z 628.061,A -85,B 0,C 180,E1 -13337.699,E2 -13337.699} C_VEL
LIN {X 0,Y 365.883,Z 617.722,A -85,B 0,C 180,E1 -13339.329,E2 -13339.329} C_VEL
LIN {X 0,Y 367.684,Z 606.027,A -85,B 0,C 180,E1 -13340.855,E2 -13340.855} C_VEL
LIN {X 0,Y 369.346,Z 593.192,A -85,B 0,C 180,E1 -13342.221,E2 -13342.221} C_VEL
LIN {X 0,Y 370.996,Z 578.803,A -85,B 0,C 180,E1 -13343.442,E2 -13343.442} C_VEL
LIN {X 0,Y 372.292,Z 564.859,A -85,B 0,C 180,E1 -13344.374,E2 -13344.374} C_VEL
LIN {X 0,Y 373.377,Z 549.274,A -85,B 0,C 180,E1 -13345.162,E2 -13345.162} C_VEL
LIN {X 0,Y 374.517,Z 530.644,A -85,B 0,C 180,E1 -13345.868,E2 -13345.868} C_VEL
LIN {X 0,Y 380.618,Z 467.141,A -85,B 0,C 180,E1 -13348.059,E2 -13348.059} C_VEL
LIN {X 0,Y 383.567,Z 439.89,A -85,B 0,C 180,E1 -13349.001,E2 -13349.001} C_VEL
LIN {X 0,Y 379.8,Z 433.399,A -85,B 0,C 180,E1 -13350.119,E2 -13350.119} C_VEL
LIN {X 0,Y 375.653,Z 427.232,A -85,B 0,C 180,E1 -13351.443,E2 -13351.443} C_VEL
LIN {X 0,Y 372.358,Z 423.031,A -85,B 0,C 180,E1 -13352.604,E2 -13352.604} C_VEL
LIN {X 0,Y 369.734,Z 419.771,A -85,B 0,C 180,E1 -13353.65,E2 -13353.65} C_VEL
LIN {X 0,Y 367.121,Z 416.645,A -85,B 0,C 180,E1 -13354.922,E2 -13354.922} C_VEL
LIN {X 0,Y 366.821,Z 415.438,A -85,B 0,C 180,E1 -13356.437,E2 -13356.437} C_VEL
LIN {X 0,Y 366.712,Z 414.455,A -85,B 0,C 180,E1 -13359.23,E2 -13359.23} C_VEL
LIN {X 0,Y 367.028,Z 414.97,A -85,B 0,C 180,E1 -13361.686,E2 -13361.686} C_VEL
LIN {X 0,Y 367.636,Z 416.162,A -85,B 0,C 180,E1 -13363.488,E2 -13363.488} C_VEL
LIN {X 0,Y 368.419,Z 417.804,A -85,B 0,C 180,E1 -13365.103,E2 -13365.103} C_VEL
LIN {X 0,Y 370.011,Z 422.06,A -85,B 0,C 180,E1 -13367.797,E2 -13367.797} C_VEL
LIN {X 0,Y 371.544,Z 426.938,A -85,B 0,C 180,E1 -13369.973,E2 -13369.973} C_VEL
LIN {X 0,Y 373.233,Z 433.621,A -85,B 0,C 180,E1 -13372.266,E2 -13372.266} C_VEL
LIN {X 0,Y 374.453,Z 439.777,A -85,B 0,C 180,E1 -13373.997,E2 -13373.997} C_VEL
LIN {X 0,Y 374.233,Z 442.479,A -85,B 0,C 180,E1 -13374.519,E2 -13374.519} C_VEL
LIN {X 0,Y 375.896,Z 455.669,A -85,B 0,C 180,E1 -13375.67,E2 -13375.67} C_VEL
LIN {X 0,Y 377.65,Z 472.798,A -85,B 0,C 180,E1 -13376.904,E2 -13376.904} C_VEL
LIN {X 0,Y 378.809,Z 488.74,A -85,B 0,C 180,E1 -13377.869,E2 -13377.869} C_VEL
LIN {X 0,Y 379.173,Z 506.724,A -85,B 0,C 180,E1 -13378.735,E2 -13378.735} C_VEL
LIN {X 0,Y 374.315,Z 570.328,A -85,B 0,C 180,E1 -13380.663,E2 -13380.663} C_VEL
LIN {X 0,Y 371.33,Z 613.844,A -85,B 0,C 180,E1 -13381.951,E2 -13381.951} C_VEL
LIN {X 0,Y 370.599,Z 622.334,A -85,B 0,C 180,E1 -13382.236,E2 -13382.236} C_VEL
LIN {X 0,Y 369.926,Z 643.105,A -85,B 0,C 180,E1 -13382.68,E2 -13382.68} C_VEL
LIN {X 0,Y 369.057,Z 657.61,A -85,B 0,C 180,E1 -13383.181,E2 -13383.181} C_VEL
LIN {X 0,Y 367.785,Z 672.672,A -85,B 0,C 180,E1 -13383.926,E2 -13383.926} C_VEL
LIN {X 0,Y 366.318,Z 687.427,A -85,B 0,C 180,E1 -13384.909,E2 -13384.909} C_VEL
LIN {X 0,Y 364.689,Z 700.249,A -85,B 0,C 180,E1 -13385.975,E2 -13385.975} C_VEL
LIN {X 0,Y 362.83,Z 713.601,A -85,B 0,C 180,E1 -13387.356,E2 -13387.356} C_VEL
LIN {X 0,Y 360.953,Z 725.741,A -85,B 0,C 180,E1 -13388.886,E2 -13388.886} C_VEL
LIN {X 0,Y 359.31,Z 736.798,A -85,B 0,C 180,E1 -13390.577,E2 -13390.577} C_VEL
LIN {X 0,Y 357.781,Z 746.099,A -85,B 0,C 180,E1 -13392.272,E2 -13392.272} C_VEL
LIN {X 0,Y 356.365,Z 755.223,A -85,B 0,C 180,E1 -13394.265,E2 -13394.265} C_VEL
LIN {X 0,Y 355.227,Z 762.788,A -85,B 0,C 180,E1 -13396.264,E2 -13396.264} C_VEL
LIN {X 0,Y 354.584,Z 768.23,A -85,B 0,C 180,E1 -13397.986,E2 -13397.986} C_VEL
LIN {X 0,Y 353.891,Z 774.133,A -85,B 0,C 180,E1 -13400.28,E2 -13400.28} C_VEL
LIN {X 0,Y 353.596,Z 777.621,A -85,B 0,C 180,E1 -13402.001,E2 -13402.001} C_VEL
LIN {X 0,Y 353.36,Z 781.164,A -85,B 0,C 180,E1 -13404.291,E2 -13404.291} C_VEL
LIN {X 0,Y 353.265,Z 783.491,A -85,B 0,C 180,E1 -13406.577,E2 -13406.577} C_VEL
LIN {X 0,Y 353.23,Z 784.659,A -85,B 0,C 180,E1 -13408.858,E2 -13408.858} C_VEL
LIN {X 0,Y 353.232,Z 784.657,A -85,B 0,C 180,E1 -13411.138,E2 -13411.138} C_VEL
LIN {X 0,Y 353.267,Z 783.482,A -85,B 0,C 180,E1 -13413.42,E2 -13413.42} C_VEL
LIN {X 0,Y 353.345,Z 781.151,A -85,B 0,C 180,E1 -13415.706,E2 -13415.706} C_VEL
LIN {X 0,Y 353.592,Z 777.609,A -85,B 0,C 180,E1 -13417.996,E2 -13417.996} C_VEL
LIN {X 0,Y 354.007,Z 772.765,A -85,B 0,C 180,E1 -13420.291,E2 -13420.291} C_VEL
LIN {X 0,Y 354.801,Z 766.485,A -85,B 0,C 180,E1 -13422.583,E2 -13422.583} C_VEL
LIN {X 0,Y 355.818,Z 758.592,A -85,B 0,C 180,E1 -13424.877,E2 -13424.877} C_VEL
LIN {X 0,Y 357.081,Z 750.163,A -85,B 0,C 180,E1 -13426.874,E2 -13426.874} C_VEL
LIN {X 0,Y 358.689,Z 739.989,A -85,B 0,C 180,E1 -13428.86,E2 -13428.86} C_VEL
LIN {X 0,Y 360.316,Z 729.563,A -85,B 0,C 180,E1 -13430.552,E2 -13430.552} C_VEL
LIN {X 0,Y 362.065,Z 718.203,A -85,B 0,C 180,E1 -13432.089,E2 -13432.089} C_VEL
LIN {X 0,Y 363.865,Z 705.826,A -85,B 0,C 180,E1 -13433.474,E2 -13433.474} C_VEL
LIN {X 0,Y 365.648,Z 692.237,A -85,B 0,C 180,E1 -13434.709,E2 -13434.709} C_VEL
LIN {X 0,Y 367.215,Z 677.952,A -85,B 0,C 180,E1 -13435.744,E2 -13435.744} C_VEL
LIN {X 0,Y 368.558,Z 663.515,A -85,B 0,C 180,E1 -13436.544,E2 -13436.544} C_VEL
LIN {X 0,Y 369.593,Z 648.399,A -85,B 0,C 180,E1 -13437.151,E2 -13437.151} C_VEL
LIN {X 0,Y 370.204,Z 634.339,A -85,B 0,C 180,E1 -13437.523,E2 -13437.523} C_VEL
LIN {X 0,Y 373.161,Z 517.433,A -85,B 0,C 180,E1 -13439.791,E2 -13439.791} C_VEL
LIN {X 0,Y 373.38,Z 504.221,A -85,B 0,C 180,E1 -13440.058,E2 -13440.058} C_VEL
LIN {X 0,Y 369.738,Z 474.933,A -85,B 0,C 180,E1 -13441.033,E2 -13441.033} C_VEL
LIN {X 0,Y 368.463,Z 465.384,A -85,B 0,C 180,E1 -13441.401,E2 -13441.401} C_VEL
LIN {X 0,Y 366.669,Z 436.95,A -85,B 0,C 180,E1 -13443.159,E2 -13443.159} C_VEL
LIN {X 0,Y 366.479,Z 432.79,A -85,B 0,C 180,E1 -13443.456,E2 -13443.456} C_VEL
LIN {X 0,Y 366.875,Z 429.605,A -85,B 0,C 180,E1 -13443.893,E2 -13443.893} C_VEL
